Universal Robots URScript: DAS428_958_02_MAR_21_DAS_lado_derecho_jig2.script

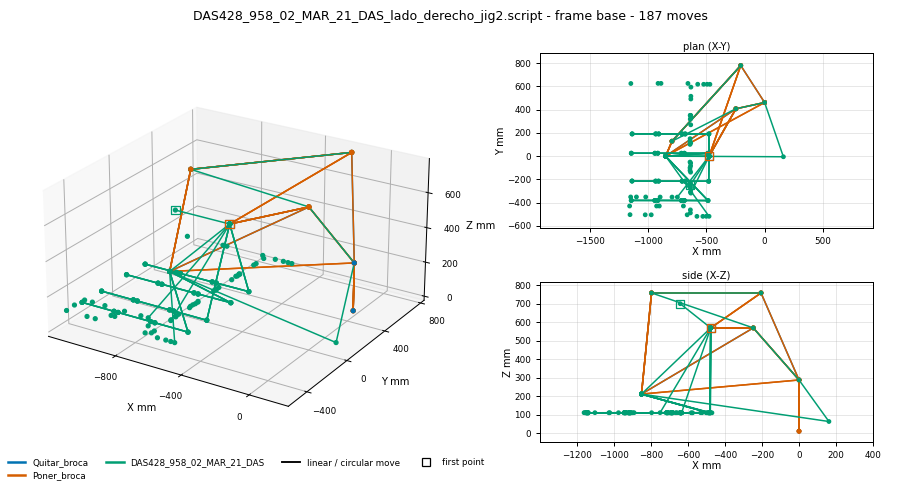
[picture p0: tool path of DAS428_958_02_MAR_21_DAS_lado_derecho_jig2.script in frame base, 187 of 840 moves have a stored position in this frame; points joined in program order, loops and branches not executed]
def DAS428_958_02_MAR_21_DAS_lado_derecho_jig2():
  set_gravity([0.0, 0.0, 9.82])
  set_standard_analog_input_domain(0, 1)
  set_standard_analog_input_domain(1, 1)
  set_tool_analog_input_domain(0, 1)
  set_tool_analog_input_domain(1, 1)
  set_analog_outputdomain(0, 0)
  set_analog_outputdomain(1, 0)
  set_input_actions_to_default()
  set_runstate_standard_digital_outputs([2])
  set_runstate_configurable_digital_outputs([1])
  set_runstate_standard_digital_output_to_value(2, 1)
  set_runstate_configurable_digital_output_to_value(1, 1)
  modbus_add_signal("192.168.10.45", 255, 187, 1, "postrnas_m187", False)
  modbus_set_signal_update_frequency("postrnas_m187", 10)
  modbus_add_signal("192.168.10.45", 255, 289, 1, "ini_cambro_m289", False)
  modbus_set_signal_update_frequency("ini_cambro_m289", 10)
  modbus_add_signal("192.168.10.45", 255, 290, 0, "fin_cambro_m290", False)
  modbus_set_signal_update_frequency("fin_cambro_m290", 10)
  modbus_add_signal("192.168.10.45", 255, 291, 1, "outputbroc_m291", False)
  modbus_set_signal_update_frequency("outputbroc_m291", 10)
  modbus_add_signal("192.168.10.45", 255, 292, 0, "fciclocarr_m292", False)
  modbus_set_signal_update_frequency("fciclocarr_m292", 10)
  modbus_add_signal("192.168.10.45", 255, 7, 1, "avancarrusel_m7", False)
  modbus_set_signal_update_frequency("avancarrusel_m7", 10)
  modbus_add_signal("192.168.10.45", 255, 252, 1, "pose2_m252", False)
  modbus_set_signal_update_frequency("pose2_m252", 10)
  modbus_add_signal("192.168.10.45", 255, 253, 1, "pose3_m253", False)
  modbus_set_signal_update_frequency("pose3_m253", 10)
  modbus_add_signal("192.168.10.45", 255, 254, 1, "pose4_m254", False)
  modbus_set_signal_update_frequency("pose4_m254", 10)
  modbus_add_signal("192.168.10.45", 255, 441, 1, "finciclo_m441", False)
  modbus_set_signal_update_frequency("finciclo_m441", 10)
  modbus_add_signal("192.168.10.45", 255, 442, 1, "finciclo_m442", False)
  modbus_set_signal_update_frequency("finciclo_m442", 10)
  modbus_add_signal("192.168.10.45", 255, 443, 1, "finciclo_m443", False)
  modbus_set_signal_update_frequency("finciclo_m443", 10)
  modbus_add_signal("192.168.10.45", 255, 503, 0, "homecobot_m503", False)
  modbus_set_signal_update_frequency("homecobot_m503", 10)
  modbus_add_signal("192.168.10.45", 255, 288, 1, "cargar_run_m288", False)
  modbus_set_signal_update_frequency("cargar_run_m288", 10)
  modbus_add_signal("192.168.10.45", 255, 287, 0, "desactiver_m288", False)
  modbus_set_signal_update_frequency("desactiver_m288", 10)
  modbus_add_signal("192.168.10.45", 255, 183, 0, "eje7home_m183", False)
  modbus_set_signal_update_frequency("eje7home_m183", 10)
  modbus_add_signal("192.168.10.45", 255, 444, 1, "finciclo_m444", False)
  modbus_set_signal_update_frequency("finciclo_m444", 10)
  modbus_add_signal("192.168.10.45", 255, 381, 0, "pat1_m381", False)
  modbus_set_signal_update_frequency("pat1_m381", 10)
  modbus_add_signal("192.168.10.45", 255, 382, 0, "pat2_m382", False)
  modbus_set_signal_update_frequency("pat2_m382", 10)
  modbus_add_signal("192.168.10.45", 255, 383, 0, "pat3_m383", False)
  modbus_set_signal_update_frequency("pat3_m383", 10)
  modbus_add_signal("192.168.10.45", 255, 384, 0, "pat4_m384", False)
  modbus_set_signal_update_frequency("pat4_m384", 10)
  modbus_add_signal("192.168.10.45", 255, 385, 0, "pat5_m385", False)
  modbus_set_signal_update_frequency("pat5_m385", 10)
  modbus_add_signal("192.168.10.45", 255, 386, 0, "pat6_m386", False)
  modbus_set_signal_update_frequency("pat6_m386", 10)
  modbus_add_signal("192.168.10.45", 255, 387, 0, "pat7_m387", False)
  modbus_set_signal_update_frequency("pat7_m387", 10)
  modbus_add_signal("192.168.10.45", 255, 388, 0, "pat8_m388", False)
  modbus_set_signal_update_frequency("pat8_m388", 10)
  modbus_add_signal("192.168.10.45", 255, 389, 0, "pat9_m389", False)
  modbus_set_signal_update_frequency("pat9_m389", 10)
  modbus_add_signal("192.168.10.45", 255, 390, 0, "pat10_m390", False)
  modbus_set_signal_update_frequency("pat10_m390", 10)
  modbus_add_signal("192.168.10.45", 255, 391, 0, "pat11_m391", False)
  modbus_set_signal_update_frequency("pat11_m391", 10)
  modbus_add_signal("192.168.10.45", 255, 392, 0, "pat12_m392", False)
  modbus_set_signal_update_frequency("pat12_m392", 10)
  modbus_add_signal("192.168.10.45", 255, 401, 0, "inipat1_m401", False)
  modbus_set_signal_update_frequency("inipat1_m401", 10)
  modbus_add_signal("192.168.10.45", 255, 402, 0, "inipat2_m402", False)
  modbus_set_signal_update_frequency("inipat2_m402", 10)
  modbus_add_signal("192.168.10.45", 255, 403, 0, "inipat3_m403", False)
  modbus_set_signal_update_frequency("inipat3_m403", 10)
  modbus_add_signal("192.168.10.45", 255, 404, 0, "inipat4_m404", False)
  modbus_set_signal_update_frequency("inipat4_m404", 10)
  modbus_add_signal("192.168.10.45", 255, 405, 0, "inipat5_m405", False)
  modbus_set_signal_update_frequency("inipat5_m405", 10)
  modbus_add_signal("192.168.10.45", 255, 406, 0, "inipat6_m406", False)
  modbus_set_signal_update_frequency("inipat6_m406", 10)
  modbus_add_signal("192.168.10.45", 255, 407, 0, "inipat7_m407", False)
  modbus_set_signal_update_frequency("inipat7_m407", 10)
  modbus_add_signal("192.168.10.45", 255, 408, 0, "inipat8_m408", False)
  modbus_set_signal_update_frequency("inipat8_m408", 10)
  modbus_add_signal("192.168.10.45", 255, 409, 0, "inipat9_m409", False)
  modbus_set_signal_update_frequency("inipat9_m409", 10)
  modbus_add_signal("192.168.10.45", 255, 410, 0, "inipat10_m410", False)
  modbus_set_signal_update_frequency("inipat10_m410", 10)
  modbus_add_signal("192.168.10.45", 255, 411, 0, "inipat11_m411", False)
  modbus_set_signal_update_frequency("inipat11_m411", 10)
  modbus_add_signal("192.168.10.45", 255, 412, 0, "inipat12_m412", False)
  modbus_set_signal_update_frequency("inipat12_m412", 10)
  modbus_add_signal("192.168.10.45", 255, 430, 0, "modeloDer_m430", False)
  modbus_set_signal_update_frequency("modeloDer_m430", 10)
  modbus_add_signal("192.168.10.45", 255, 380, 1, "mensaje_m380", False)
  modbus_set_signal_update_frequency("mensaje_m380", 10)
  modbus_add_signal("192.168.10.45", 255, 379, 0, "respues_m379", False)
  modbus_set_signal_update_frequency("respues_m379", 10)
  modbus_add_signal("192.168.10.45", 255, 251, 1, "pose1_m251", False)
  modbus_set_signal_update_frequency("pose1_m251", 10)
  modbus_set_runstate_dependent_choice("postrnas_m187",0)
  modbus_set_runstate_dependent_choice("ini_cambro_m289",0)
  modbus_set_runstate_dependent_choice("outputbroc_m291",0)
  modbus_set_runstate_dependent_choice("avancarrusel_m7",0)
  modbus_set_runstate_dependent_choice("pose2_m252",0)
  modbus_set_runstate_dependent_choice("pose3_m253",0)
  modbus_set_runstate_dependent_choice("pose4_m254",0)
  modbus_set_runstate_dependent_choice("finciclo_m441",0)
  modbus_set_runstate_dependent_choice("finciclo_m442",0)
  modbus_set_runstate_dependent_choice("finciclo_m443",0)
  modbus_set_runstate_dependent_choice("cargar_run_m288",0)
  modbus_set_runstate_dependent_choice("finciclo_m444",0)
  modbus_set_runstate_dependent_choice("mensaje_m380",0)
  modbus_set_runstate_dependent_choice("pose1_m251",0)
  set_safety_mode_transition_hardness(1)
  set_tool_communication(False, 115200, 0, 1, 1.5, 3.5)
  set_tool_output_mode(0)
  set_tool_digital_output_mode(0, 1)
  set_tool_digital_output_mode(1, 1)
  set_tool_voltage(0)
  set_tcp(p[4.109330471764039E-4,-0.21829828276152607,0.037994196120996,1.5580092985761962,-0.12546870791316503,0.12120248426608284])
  set_payload(1.5)
  step_count_e0f46a76_adf3_4eac_87f0_1f0dabebea5e = 0
  thread Step_Counter_Thread_08bb6925_5529_4cdb_99f9_8a05e79ee4da():
    while (True):
      step_count_e0f46a76_adf3_4eac_87f0_1f0dabebea5e = step_count_e0f46a76_adf3_4eac_87f0_1f0dabebea5e + 1
      sync()
    end
  end
  run Step_Counter_Thread_08bb6925_5529_4cdb_99f9_8a05e79ee4da()
  global contador=0
  global i_var_1=0
  global Pallet_1_cnt_1=1
  global Pallet_1_cnt=1
  global Line_1=p[0.0,0.0,0.0,0.0,0.0,0.0]
  global Line_2=p[0.0,0.0,0.0,0.0,0.0,0.0]
  global Line_3=p[0.0,0.0,0.0,0.0,0.0,0.0]
  global Line_4=p[-0.2932874787951964,0.3932288129452105,0.013749459185886714,0.019478391032120013,-0.0350876085014595,1.5300278925331599]
  global Line_5=p[0.0,0.0,0.0,0.0,0.0,0.0]
  global Plane_1=p[-0.4357649673792705,0.3571224276764373,-0.011331751409534768,-0.03455953496512708,-0.012487423981114925,3.103751116092306]
  global Plane_2=p[-0.4823864034329737,0.3302516442079689,0.014283714098506706,0.017125077458443067,0.05770060098903715,-2.9134709732588786]
  global Plane_3=p[0.003678615545088639,0.4082921331082374,0.10477407557236007,-2.072177303174012E-4,7.379081343290108E-4,-6.424400645467977E-4]
  global Plane_4=p[-0.4500206307677429,-0.2823718146925442,-0.4767416657426552,0.013278190059218174,0.013334473770785706,1.8479691991032237]
  global Plano_patron1=p[-0.7699005610122596,0.304894434078545,0.0420369514744936,-0.0031270356010209216,1.7180543614697593E-4,-3.508888786211572E-5]
  global Point_13=p[0.0,0.0,0.0,0.0,0.0,0.0]
  global Point_3=p[0.0,0.0,0.0,0.0,0.0,0.0]
  global Point_8=p[0.0,0.0,0.0,0.0,0.0,0.0]
  global Punto_prot_1=p[0.0,0.0,0.0,0.0,0.0,0.0]
  global Punto_seg_der=p[0.23741638234469645,0.3587772222537799,0.42419077585740217,0.818517054876345,1.4216436941132238,1.005041187710707]
  global pisp_958=p[-0.41395442210486977,-0.2082168853247176,0.041553466664982,0.014014788518713659,0.01101911827984854,1.569193423241601]
  rtde_set_watchdog("speed_slider_mask", 10.0, "ignore")
  global Traslacion_p=p[-.641047005341, -.250866212824, .699550653028, 2.557164228531, -1.705634893075, -.146977311260]
  global Traslacion_q=[-0.008123397867477067, -1.6493627997444174, 1.2335318981093104, 0.31142302236535, -5.2726714898139235, -0.002836317283104961]
  global Home2_p=p[-.476229469061, .000000001191, .568736718299, 2.026271312133, -2.392905827360, -.020822003949]
  global Home2_q=[-0.5681294612478887, -2.032770910737735, 1.7176337322759885, 0.3114230223653604, -5.272671489814012, -0.002836317283105849]
  global Home3_p=p[-.850182153427, -.000000001054, .211319941039, -2.029706048810, 2.396843749609, .006593444086]
  global Home3_q=[-0.2508712563283524, -1.32118636682587, 1.7236419957383333, -0.39530717300436535, -4.957384713543316, -0.003346356527782035]
  global Home4_p=p[-.850182153426, -.000000001054, .211319941039, -2.029706048810, 2.396843749609, .006593444086]
  global Home4_q=[-0.25087125632834173, -1.32118636682587, 1.7236419957383335, -0.39530717300436535, -4.957384713543306, -0.003346356527782035]
  global PosicionApagado_p=p[.162342971637, -.004968702407, .063230450635, -1.839175988951, .225343983922, .171657948894]
  global PosicionApagado_q=[1.570738988136085, -1.5704867605983486, 2.609644234392225, 0.2613772922410976, -4.625127484032603, 1.7781079770353217E-5]
  global Precambio_broca_p=p[.000830370305, .461517540512, .287521124194, -.221784750204, -3.131955254916, .000429460883]
  global Precambio_broca_q=[-2.1838225298159477, -2.0964618902985066, 2.243453456263678, -0.13436505871461257, -5.342774534909408, -0.004043449473680738]
  global yendo1_p=p[-.246136658478, .407690142824, .568736718299, -.589365823667, 3.084367220712, .022757599334]
  global yendo1_q=[-1.5957647560042467, -2.0327709107377157, 1.7176337322759783, 0.31142302236534997, -5.272671489813924, -0.002836317283104961]
  global Precam_bro1_p=p[-.795770836809, .128511169110, .757632075886, 1.553391881516, -2.198703969583, -.808866164734]
  global Precam_bro1_q=[-0.42509351308843435, -1.7320527113687803, 1.4689329310980348, -0.39530717300436535, -4.957384713543306, -0.003346356527782035]
  global Precam_bro2_p=p[-.204472177612, .779716277811, .757632075886, -.111446445846, 2.933975892584, 1.018360754732]
  global Precam_bro2_q=[-1.5793151587200072, -1.7320527113687803, 1.4689329310980348, -0.39530717300436535, -4.957384713543306, -0.003346356527782035]
  global Linea1_A_p=p[-.480065223067, -.215566781041, .110154596536, 2.026283817979, -2.392895080548, -.020829635760]
  global Linea1_A_q=[0.12579830563919536, -1.756524695513292, 2.3832893788943412, -0.6314317143827912, -4.58099271090342, -0.0047002730467511356]
  global Linea1_B_p=p[-.683259997836, -.215006380581, .110473377935, 2.026330825697, -2.392937749126, -.020814905630]
  global Linea1_B_q=[0.07860269075896831, -1.433097350639013, 2.069317086211182, -0.6407207629147003, -4.628316962573399, -0.00423059265382264]
  global Linea1_C_p=p[-.708659998696, -.214985847345, .110510820529, 2.026397919151, -2.392909525922, -.020800557194]
  global Linea1_C_q=[0.07508702140477563, -1.3964952588668957, 2.0250632394702635, -0.6330397547175677, -4.631871660537247, -0.004203657105243508]
  global Linea1_D_p=p[-.911541589269, -.214532502479, .110305804030, 2.026334474712, -2.392925442770, -.020895674247]
  global Linea1_D_q=[0.054901387986126586, -1.113040084501037, 1.6299948744075297, -0.5214573164063481, -4.651846197735423, -0.004103335395922336]
  global Linea1_E_p=p[-.936517713267, -.214589312402, .110514758557, 2.026299167222, -2.392914652900, -.020910067647]
  global Linea1_E_q=[0.053256694947611545, -1.0779791152787563, 1.5748557207640133, -0.5014068860788594, -4.65343899925324, -0.0040886755584823575]
  global Linea1_F_p=p[-1.139513888655, -.213880830394, .110127483913, 2.026321929742, -2.392901637414, -.020934114652]
  global Linea1_F_q=[0.04170148606385503, -0.7616832269463547, 1.037979133577118, -0.2808209912067561, -4.664495303417296, -0.0041165609944391335]
  def calculate_point_to_move_towards(feature, direction, position_distance):
    local posDir=[direction[0], direction[1], direction[2]]
    if (norm(posDir) < 1e-6):
      return get_target_waypoint()
    end
    local direction_vector_normalized=normalize(posDir)
    local displacement_pose=p[direction_vector_normalized[0] * position_distance,direction_vector_normalized[1] * position_distance,direction_vector_normalized[2] * position_distance,0,0,0]
    local wanted_displacement_in_base_frame=pose_sub(pose_trans(feature, displacement_pose), feature)
    return pose_add(get_target_waypoint(), wanted_displacement_in_base_frame)
  end
  global Linea2_A_p=p[-.478569784260, .191006236121, .110522539661, 2.026309184484, -2.392844209472, -.020866358396]
  global Linea2_A_q=[-1.0119726055803717, -1.7923449463408154, 2.4087968238915316, -0.622613470734211, -5.718752417482761, 0.0017055247889921077]
  global Linea2_B_p=p[-.681936431684, .191001701528, .110452389888, 2.026254746254, -2.392870981141, -.020856049736]
  global Linea2_B_q=[-0.660932087342812, -1.45042632220569, 2.089702129115615, -0.644100890415773, -5.3678371124098305, -6.551765912714558E-4]
  global Linea2_C_p=p[-.707213860547, .190994877950, .110602621396, 2.026215373389, -2.392855024802, -.020833229234]
  global Linea2_C_q=[-0.6329633221322801, -1.4131450476618888, 2.0452127395946604, -0.63685969915739, -5.339852460491649, -7.508873236439229E-4]
  global Linea2_D_p=p[-.910191818076, .191478760022, .110348317855, 2.026197382673, -2.392838381909, -.020850455695]
  global Linea2_D_q=[-0.47159299446006386, -1.1248659495364315, 1.6481441269090888, -0.5278387233410813, -5.17831767767195, -0.0015522613841945088]
  global Linea2_E_p=p[-.935619999730, .191518537756, .110453838050, 2.026145948950, -2.392831929254, -.020993754227]
  global Linea2_E_q=[-0.45687914266405194, -1.088905585645314, 1.5922022218243828, -0.5079352095297214, -5.1635430614079825, -0.0016331567764398258]
  global Linea2_F_p=p[-1.138394848852, .191499459928, .110212234352, 2.026158962848, -2.392763937758, -.020990642855]
  global Linea2_F_q=[-0.36535169690146674, -0.7732464559921581, 1.0587228640233546, -0.29003791508182974, -5.071546930507635, -0.0021173024104594873]
  global Linea7_A_p=p[-.749560809058, -.351839418109, .110842549516, 3.108416959288, -.375864319326, -.017387250007]
  global Linea7_A_q=[0.03345458497850107, -1.1510417746331125, 1.685959359828983, -0.5377045142036341, -6.168946681556185, -0.005399210077573713]
  global Linea7_B_p=p[-.795370452792, -.351638127396, .110748062148, 3.108426240568, -.375794652077, -.017394126552]
  global Linea7_B_q=[0.031278459806111415, -1.0863508926378662, 1.5866056594622966, -0.5030470097495243, -6.17110138542474, -0.0053959734286266325]
  global Linea8_A_p=p[-.897664645372, -.351420839665, .110405519513, 3.108418537152, -.375848167267, -.017413606898]
  global Linea8_A_q=[0.0274697684633054, -0.9358640938182816, 1.3416002369808222, -0.4084067160106146, -6.174672123664049, -0.005526846744682956]
  global Linea8_B_p=p[-1.021742815617, -.350913421148, .110769725780, 3.108429042178, -.375802310169, -.017313462884]
  global Linea8_B_q=[0.023588010639285104, -0.727028660928073, 0.9730136327156043, -0.24827020482455175, -6.178185664503821, -0.005846159791357053]
  global Linea9_A_p=p[-1.101640143677, -.350630386336, .110828130197, 3.108414048814, -.375882576694, -.017444590769]
  global Linea9_A_q=[0.021544403730552553, -0.5492801598617163, 0.6399908213108159, -0.09279065312938162, -6.179741333586448, -0.006134404310005337]
  global Linea9_B_p=p[-1.151201662491, -.350816300328, .110404811963, 3.108409734650, -.375889963226, -.017367079724]
  global Linea9_B_q=[0.020666902118270467, -0.3678660308533921, 0.2849675943410323, 0.08068312139155243, -6.180088831683512, -0.005949069824949582]
  global Linea10_A_p=p[-.633308011674, -.317691120510, .110994505067, 3.108412257751, -.375924840358, -.017335462218]
  global Linea10_A_q=[-0.015400976327146765, -1.3286836616185038, 1.936773774913373, -0.6125541680104964, -6.2178811871620026, -0.0036320224430834713]
  global Linea10_B_p=p[-.636723959746, -.266696422603, .110313777239, 2.020474030001, -2.393914578871, -.020559556678]
  global Linea10_B_q=[0.1863095606962153, -1.4646980412767157, 2.1071523959293508, -0.6494023099187478, -4.517372761756647, -0.0030763184180990777]
  global Linea11_A_p=p[-.635968117082, -.137768266518, .110291503345, 2.022156502066, -2.396023902726, -.017001304800]
  global Linea11_A_q=[-0.07354604755883543, -1.5471079384277004, 2.1956073198093513, -0.6515202395877564, -4.777150906045714, -0.0016328727799539422]
  global Linea11_B_p=p[-.635823762501, -.083112159886, .110947967545, 2.020383801711, -2.393902625595, -.020556219708]
  global Linea11_B_q=[-0.1908380759122572, -1.5708643495776826, 2.219519946363693, -0.6552069469693311, -4.894453843584338, -5.759924145127826E-4]
  global Linea12_A_p=p[-.635349004319, -.059560123377, .110675436750, 2.020448494290, -2.393915459802, -.020549325419]
  global Linea12_A_q=[-0.2417163087330083, -1.5775265863609773, 2.226737904634896, -0.6557292375944215, -4.945355909075068, -2.7983922817842455E-4]
  global Linea12_B_p=p[-.634712541835, .114180549607, .110553374724, 2.020445364866, -2.393872518012, -.020639369641]
  global Linea12_B_q=[-0.5920002980493377, -1.5626330075993593, 2.212116743928059, -0.656716518252761, -5.2956538993562265, 0.0023497530147947032]
  global Linea13_A_p=p[-.634623456483, .269837596517, .110201600077, 2.020453398687, -2.393912519416, -.020625959570]
  global Linea13_A_q=[-0.8324062816272679, -1.467834151680524, 2.1109901381841176, -0.6517507900808974, -5.53605704845582, 0.004880071949341591]
  global Linea13_B_p=p[-.634042726961, .326314422350, .110496359725, 2.020453146279, -2.393880944182, -.020556436265]
  global Linea13_B_q=[-0.9013131509490719, -1.4220878936638712, 2.0569245075861637, -0.6440785774915501, -5.604971402017175, 0.005892023416525838]
  global Linea14_A_p=p[-.633962563051, .349886895745, .111384319105, 2.020461054934, -2.393837815408, -.020488388436]
  global Linea14_A_q=[-0.9271552684385451, -1.4021744596762797, 2.030901915913411, -0.638246246484969, -5.630828387156736, 0.006335596407090804]
  global Linea14_B_p=p[-.633710645144, .491847819742, .110684020249, 2.020465968208, -2.393853523670, -.020498328553]
  global Linea14_B_q=[-1.0540906694923677, -1.2626852057640106, 1.849914655177884, -0.5986568379003074, -5.757703248039979, 0.008776098960622295]
  global Linea15_A_p=p[-.633318381480, .515440368134, .110157981608, 2.020364155203, -2.393955709596, -.020508500424]
  global Linea15_A_q=[-1.0716567160130523, -1.2377525992845975, 1.8159966720140375, -0.590008690959742, -5.775162769690162, 0.009175048989259693]
  global Linea15_B_p=p[-.632970544234, .593971386241, .110611257026, 2.020441893491, -2.393867996682, -.020560033230]
  global Linea15_B_q=[-1.122474592013197, -1.1525133394351883, 1.6903287270969671, -0.5508046641787523, -5.825981972795807, 0.0105832391144433]
  global Linea16_A_p=p[-.469658501632, .618240146447, .110222995954, -.214451812264, -3.127782132936, -.004019473137]
  global Linea16_A_q=[-1.0558229732465527, -1.3016284898486745, 1.9002200310933528, -0.5927846748758361, -4.220581777772279, 0.011476321502457587]
  global Linea16_B_p=p[-.493719050069, .618586170158, .110182854162, -.214521728939, -3.127775191063, -.003963807283]
  global Linea16_B_q=[-1.0238267857309111, -1.275874279860929, 1.8652664634035965, -0.5834704347683779, -4.1885285819385825, 0.011722546182054927]
  global Linea17_A_p=p[-.523228961738, .618283097935, .110575467666, -.214471054905, -3.127807816993, -.003922935561]
  global Linea17_A_q=[-0.986020922475106, -1.2448369572559947, 1.8212231475782765, -0.570331686133752, -4.150737151059812, 0.011980907174432787]
  global Linea17_B_p=p[-.574504951156, .618780338898, .110128214767, -.214469703842, -3.127802767109, -.003936726452]
  global Linea17_B_q=[-0.9261028235589457, -1.187335623873139, 1.739319222569904, -0.5457499909581429, -4.090780405906422, 0.012429946919677803]
  global Linea18_A_p=p[-.658632612166, .625710002031, .110712740654, -.214452471617, -3.127789736506, -.003965415657]
  global Linea18_A_q=[-0.845178287049178, -1.0844314603972958, 1.5815647493127447, -0.49060909462111013, -4.009765233293088, 0.013074519407750586]
  global Linea18_AB_p=p[-.890202921445, .626113814922, .110875277310, -.214452404345, -3.127789769971, -.003965502225]
  global Linea18_AB_q=[-0.666410313611312, -0.7691628241018513, 1.0473212163579504, -0.27060302401380376, -3.8304915682302414, 0.014782791955626706]
  global Linea18_BA_p=p[-.915681226687, .626148241580, .110663930708, -.214452382992, -3.127789782522, -.003965540155]
  global Linea18_BA_q=[-0.6508504262668842, -0.7263239276067006, 0.9700203563697315, -0.2360215468567155, -3.814840986504011, 0.014958594137021445]
  global Linea18_B_p=p[-1.149588289356, .625184723765, .110393131864, 1.164105535838, -2.905778629907, .010490328627]
  global Linea18_B_q=[-0.6326303647503142, -0.3275146210078148, 0.20111537186222211, 0.13508347000242882, -4.694571332776312, 0.015612052511970474]
  global Linea3_A_p=p[-.486113587685, -.381654790172, .110209853748, -2.029718171558, 2.396836025242, .006539356697]
  global Linea3_A_q=[0.5023501146744431, -1.5361328198955349, 2.1811298091833677, -0.6380602103615596, -4.2045801543318735, 0.0021335806977313965]
  global Linea3_B_p=p[-.689309999510, -.380790560286, .110221298638, -2.029741328186, 2.396866665706, .006544867438]
  global Linea3_B_q=[0.3500483409555937, -1.2996119924085647, 1.897164714326017, -0.5909098707750893, -4.3568479224424745, 0.0011255087267496577]
  global Linea3_C_p=p[-.714729999690, -.381227126176, .110547071161, -2.029776929873, 2.396879295064, .006534577602]
  global Linea3_C_q=[0.33744999495907063, -1.2688250546952826, 1.8544576378801096, -0.5790270771094068, -4.369441028028362, 0.0010604390539933767]
  global Linea3_D_p=p[-.917837219491, -.380541767460, .110221865782, -2.029755394743, 2.396894821329, .006515015900]
  global Linea3_D_q=[0.2571038234470917, -1.0113929982879881, 1.4652198238047056, -0.44729400411425146, -4.449521148440042, 5.150299017975257E-4]
  global Linea3_E_p=p[-.943229998544, -.380750053929, .110259990709, -2.029745434063, 2.396926573302, .006499247846]
  global Linea3_E_q=[0.2498513013118595, -0.9766011167360098, 1.4078530008671004, -0.42473280670143687, -4.4567064172282045, 4.774193732002274E-4]
  global Linea3_F_p=p[-1.146085092422, -.380439604703, .110221400844, -2.029733453251, 2.396965844598, .006565203868]
  global Linea3_F_q=[0.2019713672814234, -0.646294758886178, 0.8226722249789473, -0.16994117112115248, -4.503916586459291, 6.524146887532112E-5]
  global Linea4_A_p=p[-.486108757094, .025046304243, .110758143818, -2.029716299014, 2.396836938000, .006515392677]
  global Linea4_A_q=[-0.6198243103301522, -1.8882999158352325, 2.4675810378541345, -0.5700854657560619, -5.326458533546596, -0.006784361427073726]
  global Linea4_B_p=p[-.689317790597, .025343044299, .110270277143, -2.029778955477, 2.396879909406, .006610652550]
  global Linea4_B_q=[-0.3753982057274481, -1.4863250332384972, 2.127234561670928, -0.6334691626908935, -5.0823254476145046, -0.003953878004303135]
  global Linea4_C_p=p[-.714720878933, .025085639180, .110564947322, -2.029759600612, 2.396870390258, .006543964992]
  global Linea4_C_q=[-0.3574732421871216, -1.4458978723273388, 2.0805072777503337, -0.62720153470989, -5.064395308840017, -0.0037851685217935582]
  global Linea4_D_p=p[-.918062834429, .025352519761, .110171259010, -2.029799128046, 2.396930392653, .006486194650]
  global Linea4_D_q=[-0.2611086455128149, -1.1428166917109337, 1.6724418329476345, -0.5225904730037927, -4.9678804000226116, -0.0028991485058149635]
  global Linea4_E_p=p[-.942590633843, .025362358338, .110649521713, -2.029804551742, 2.396899081770, .006457624074]
  global Linea4_E_q=[-0.25289441014648517, -1.1074268163516194, 1.6172408610903544, -0.5027734532907475, -4.9596442412571164, -0.002849666115224636]
  global Linea4_F_p=p[-1.145809999790, .025560776894, .110408083890, -2.029813008116, 2.396940383966, .006563150563]
  global Linea4_F_q=[-0.20084306122313045, -0.7863624812136436, 1.078794535602439, -0.2855892759874594, -4.907083004154831, -0.00254582608889109]
  global Linea19_A_p=p[-.476993752079, -.517247348420, .110482180983, 3.111546112853, -.391923915264, .008397312856]
  global Linea19_A_q=[0.3663200128941275, -1.4014222930595945, 2.0287178354256366, -0.6180541023023682, -5.826341631139508, -1.5291289902208405E-4]
  global Linea19_B_p=p[-.500828906079, -.517140718168, .110478451867, 3.111546096446, -.391923927944, .008397321867]
  global Linea19_B_q=[0.35160318977889826, -1.372483224500158, 1.9927968502195714, -0.6107942241264501, -5.841051456629851, -4.441148050489119E-4]
  global Linea20_A_p=p[-.530365704390, -.517559293263, .110808466240, 3.111546095803, -.391923919730, .008397321765]
  global Linea20_A_q=[0.33563033058992797, -1.3363269605580115, 1.94574379450221, -0.5995698399171738, -5.857010959106091, -7.866311909552337E-4]
  global Linea20_B_p=p[-.581158312152, -.517498500963, .110403002315, 3.111546108155, -.391923880414, .008397313958]
  global Linea20_B_q=[0.3100718063294732, -1.2734435128638637, 1.862269700997377, -0.5783990031154378, -5.8825402788566326, -0.0013910864741042417]
  global Linea21_A_p=p[-.665124494580, -.504210865882, .110600214775, 3.111546096026, -.391923862954, .008397317428]
  global Linea21_A_q=[0.2573690543360489, -1.1776890584644226, 1.7249145049026704, -0.5352634869878585, -5.935170767510868, -0.002981287852510839]
  global Linea21_AB_p=p[-.974251236041, -.504210865628, .110800066306, 3.111546114034, -.391923818122, .008397307719]
  global Linea21_AB_q=[0.1799298970176908, -0.7275076895770098, 0.9726424894081029, -0.22955136462346193, -6.011907604967895, -0.006694782410928468]
  global Linea21_BA_p=p[-1.025948854959, -.504193334254, .110365518030, 3.111461951708, -.391950297460, .007971986720]
  global Linea21_BA_q=[0.1711561465100031, -0.6245380104555593, 0.7826065934061077, -0.14219863176293934, -6.020415742618897, -0.00727529467707555]
  global Linea21_B_p=p[-1.156707649875, -.503072794545, .110552345697, -2.509967435901, 1.875250959640, .002018781675]
  global Linea21_B_q=[0.24820218748779244, -0.5254029363972528, 0.5900463054518754, -0.04848122613311023, -4.910307707512297, -0.005929498886956708]
  global Linea22_A_p=p[-.637632433174, -.487982976479, .110979882815, 3.111546090028, -.391923816497, .008397315714]
  global Linea22_A_q=[0.24472934312467132, -1.2243225409022536, 1.7920552918632602, -0.5553129495014248, -5.947844161109764, -0.0034535219061346822]
  global Linea22_B_p=p[-.637632431354, -.461705375702, .110442752941, 3.111546036492, -.391923771717, .008397328631]
  global Linea22_B_q=[0.20717345223233252, -1.241126788140571, 1.8170870077379373, -0.5619896731518628, -5.985409130317459, -0.0050445535333150104]
  global Linea23_A_p=p[-.637534615339, -.308489261992, .110677052130, 3.111545937941, -.391923740021, .008397338509]
  global Linea23_A_q=[-0.028811057420131903, -1.3103407381530268, 1.9122910134814681, -0.5347248377646263, -6.221285712923422, -0.05854924353866764]
  global Linea23_B_p=p[-.640733962739, -.257360958137, .110320484628, -1.919417494801, 2.483289836721, .006037999405]
  global Linea23_B_q=[0.1905486224517663, -1.450436264205365, 2.0857635636442016, -0.6270384051172089, -4.427102446372631, -1.2154783732398755E-4]
  global Linea24_A_p=p[-.640733961490, -.233284408478, .110638871698, -1.919417552760, 2.483289783731, .006038056909]
  global Linea24_A_q=[0.14545722065475164, -1.4688531178545041, 2.1062141334115556, -0.629125928981761, -4.472191088464225, -5.194241954580292E-4]
  global Linea24_B_p=p[-.640733960275, -.122850233085, .110748525345, -1.919417597211, 2.483289752526, .006038102658]
  global Linea24_B_q=[-0.07605491895077954, -1.5353858090675878, 2.1786254928410287, -0.6349982171419359, -4.693686238133267, -0.0024004120313705357]
  global Linea25_A_p=p[-.640733959025, -.099756217052, .110149053398, -1.919417622933, 2.483289733447, .006038127253]
  global Linea25_A_q=[-0.1244406410731358, -1.544441361062633, 2.189369992241023, -0.6366292245286829, -4.742070057375175, -0.0028048012168682135]
  global Linea25_B_p=p[-.640733958354, -.050488778220, .110217684856, -1.919417690989, 2.483289674763, .006038178959]
  global Linea25_B_q=[-0.2283127239691316, -1.5597473241762696, 2.204914426396905, -0.6366747472205034, -4.845933707721189, -0.003691692902822119]
  global Linea26_A_p=p[-.640547506113, .101329564039, .110865193067, -1.919417715349, 2.483289689335, .006038198474]
  global Linea26_A_q=[-0.5332933914937019, -1.5549547991705772, 2.1986195220763918, -0.6339933161425408, -5.150899742746004, -0.006567092346116965]
  global Linea26_B_p=p[-.640680925269, .126812188772, .110399195482, -1.919417776128, 2.483289636172, .006038228077]
  global Linea26_B_q=[-0.5793189919827881, -1.5454213815793807, 2.1898401188412677, -0.6344739078467976, -5.196927100374702, -0.007060981198389271]
  global Linea27_A_p=p[-.640020451439, .150733100880, .110213160527, -1.919417813264, 2.483289585399, .006038241789]
  global Linea27_A_q=[-0.6217233925628083, -1.536230558235598, 2.180685216451952, -0.6342282470711922, -5.2393319968885415, -0.007541218547958195]
  global Linea27_B_p=p[-.638705853179, .318073094658, .110644167614, .116299088145, 3.121658150077, .005213984395]
  global Linea27_B_q=[-0.5302181957807237, -1.311893423219579, 1.9124676839697672, -0.5889762150838447, -3.75724236079801, -0.005733470438864963]
  global Linea28_B_p=p[-.638705854413, .351254438579, .110847636331, .116299139192, 3.121658163812, .005213903305]
  global Linea28_B_q=[-0.5749160295300664, -1.298447915414732, 1.8940103653434506, -0.5845949761528715, -3.801930405986168, -0.006576175916428895]
  global Linea29_A_p=p[-.697641532877, -.428593360272, .109990008742, -2.801724319039, 1.417160453684, .007198341972]
  global Linea29_A_q=[0.23527656453246326, -1.2789397769027335, 1.8687632760476625, -0.5784646150523693, -5.271258681648637, -0.008392583459158942]
  global Linea29_AB_p=p[-.904922459205, -.428636744368, .110456720257, -2.801724313385, 1.417160441963, .007198353879]
  global Linea29_AB_q=[0.17841388372429012, -1.0033716864184807, 1.4509125680551742, -0.43568055422700613, -5.327850178749621, -0.009190677590165564]
  global Linea29_BA_p=p[-.927926651083, -.428699716140, .110396892952, -2.803374774073, 1.417906295507, .010979680109]
  global Linea29_BA_q=[0.1737614027292249, -0.9719074952973319, 1.3997777298545344, -0.41899622204942855, -5.332520268083923, -0.0092330916124439]
  global Linea29_B_p=p[-1.160230525221, -.428650841833, .110797243179, -2.801724280945, 1.417160425039, .007198392254]
  global Linea29_B_q=[0.1368429869194676, -0.5546997699196048, 0.6476482713797873, -0.08061893151237864, -5.368496825996519, -0.009905759515234536]
  global Dejar_broca_p=p[.000823895285, .461515686418, .010824983886, -.221812507768, -3.131977618886, .000372128741]
  global Dejar_broca_q=[-2.183487269545523, -1.7626289818446779, 2.619089631151862, -0.8448915610823917, -5.34389996121201, -0.0023222697552238714]
  def Quitar_broca():
    $ 5362 "Quitar_broca" "noBreak"
    $ 5363 "Quitar_broca"
    $ 5364 "barrenos_hechos≔barrenos_hechos+1"
    global barrenos_hechos=barrenos_hechos+1
    $ 5371 "If barrenos_hechos≟14 or cambiar_broca≟ True "
    if (barrenos_hechos == 14  or  cambiar_broca ==   True  ):
      $ 5372 "'Codigo de quitar broca'"
      # 'Codigo de quitar broca'
      $ 5373 "MoveL"
      $ 5374 "Direction: Base Z+"
      global move_thread_flag_5374=0
      thread move_thread_5374():
        enter_critical
        move_thread_flag_5374 = 1
        local towardsPos=calculate_point_to_move_towards(p[0.0,0.0,0.0,0.0,0.0,0.0], [0.0,0.0,1.0], 0.05)
        movel(towardsPos, a=1.2, v=0.25)
        move_thread_flag_5374 = 2
        exit_critical
      end
      move_thread_flag_5374 = 0
      move_thread_han_5374 = run move_thread_5374()
      while (True):
        sleep(1.0E-10)
        if (move_thread_flag_5374 > 1):
          join move_thread_han_5374
          $ 5375 "Until (distance)"
          break
        end
        sync()
      end
      $ 5376 "If eje7≟2"
      if (eje7 == 2):
        $ 5377 "Home2" "breakAfter"
        movel(Home2_p, a=1.2, v=0.25)
        $ 5378 "yendo1" "breakAfter"
        movel(yendo1_p, a=1.2, v=0.25)
      end
      $ 5379 "If eje7≟3"
      if (eje7 == 3):
        $ 5380 "Home3" "breakAfter"
        movel(Home3_p, a=1.2, v=0.25)
        $ 5381 "Precam_bro1" "breakAfter"
        movel(Precam_bro1_p, a=1.2, v=0.25)
        $ 5382 "Precam_bro2" "breakAfter"
        movel(Precam_bro2_p, a=1.2, v=0.25)
      end
      $ 5383 "Precambio_broca" "breakAfter"
      movel(Precambio_broca_p, a=1.2, v=0.25)
      $ 5384 "Dejar_broca" "breakAfter"
      movel(Dejar_broca_p, a=0.1, v=0.09)
      $ 5385 "Set outputbroc_m291=Encender"
      modbus_set_output_signal("outputbroc_m291", True)
      $ 5386 "Wait: 2.0"
      sleep(2.0)
      $ 5388 "Wait: 2.0"
      sleep(2.0)
      $ 5389 "Set outputbroc_m291=Apagar"
      modbus_set_output_signal("outputbroc_m291", False)
      $ 5390 "Wait: 0.5"
      sleep(0.5)
      $ 5391 "Wait fciclocarr_m292=LO"
      while (modbus_get_signal_status("fciclocarr_m292") == True):
        sync()
      end
      $ 5392 "Wait: 0.5"
      sleep(0.5)
      $ 5394 "MoveL"
      $ 5395 "Precambio_broca" "breakAfter"
      movel(Precambio_broca_p, a=0.1, v=0.09)
      $ 5396 "Set avancarrusel_m7=Encender"
      modbus_set_output_signal("avancarrusel_m7", True)
      $ 5397 "Wait: 2.0"
      sleep(2.0)
      $ 5398 "Set avancarrusel_m7=Apagar"
      modbus_set_output_signal("avancarrusel_m7", False)
      $ 5399 "Wait: 0.1"
      sleep(0.1)
    end
  end
  def Poner_broca():
    $ 5400 "Poner_broca" "noBreak"
    $ 5401 "Poner_broca"
    $ 5402 "If cambiar_broca≟ True  or iniciando_prog≟ True "
    if (cambiar_broca ==   True    or  iniciando_prog ==   True  ):
      $ 5403 "'Codigo de poner broca'"
      # 'Codigo de poner broca'
      $ 5404 "Set ini_cambro_m289=Apagar"
      modbus_set_output_signal("ini_cambro_m289", False)
      $ 5405 "MoveL"
      $ 5406 "If eje7≟2 and iniciando_prog≟ True "
      if (eje7 == 2  and  iniciando_prog ==   True  ):
        $ 5407 "Home2" "breakAfter"
        movel(Home2_p, a=1.2, v=0.25)
        $ 5408 "yendo1" "breakAfter"
        movel(yendo1_p, a=1.2, v=0.25)
      end
      $ 5409 "If eje7≟3 and iniciando_prog≟ True "
      if (eje7 == 3  and  iniciando_prog ==   True  ):
        $ 5410 "Home3" "breakAfter"
        movel(Home3_p, a=1.2, v=0.25)
        $ 5411 "Precam_bro1" "breakAfter"
        movel(Precam_bro1_p, a=1.2, v=0.25)
        $ 5412 "Precam_bro2" "breakAfter"
        movel(Precam_bro2_p, a=1.2, v=0.25)
      end
      $ 5413 "Precambio_broca" "breakAfter"
      movel(Precambio_broca_p, a=1.2, v=0.25)
      $ 5414 "Popup: Cambia a las siguientes brocas"
      popup("Cambia a las siguientes brocas", "Advertencia", True, False, blocking=True)
      $ 5415 "Dejar_broca" "breakAfter"
      movel(Dejar_broca_p, a=0.1, v=0.09)
      $ 5416 "Set ini_cambro_m289=Encender"
      modbus_set_output_signal("ini_cambro_m289", True)
      $ 5417 "Wait: 2.0"
      sleep(2.0)
      $ 5419 "Wait: 2.0"
      sleep(2.0)
      $ 5420 "Set ini_cambro_m289=Apagar"
      modbus_set_output_signal("ini_cambro_m289", False)
      $ 5421 "Wait: 0.5"
      sleep(0.5)
      $ 5422 "Wait fciclocarr_m292=LO"
      while (modbus_get_signal_status("fciclocarr_m292") == True):
        sync()
      end
      $ 5423 "Wait: 0.5"
      sleep(0.5)
      $ 5425 "MoveL"
      $ 5426 "Precambio_broca" "breakAfter"
      movel(Precambio_broca_p, a=0.1, v=0.09)
      $ 5427 "If eje7≟2"
      if (eje7 == 2):
        $ 5428 "yendo1" "breakAfter"
        movel(yendo1_p, a=1.2, v=0.25)
        $ 5429 "Home2" "breakAfter"
        movel(Home2_p, a=1.2, v=0.25)
      end
      $ 5430 "If eje7≟3"
      if (eje7 == 3):
        $ 5431 "Precam_bro2" "breakAfter"
        movel(Precam_bro2_p, a=1.2, v=0.25)
        $ 5432 "Precam_bro1" "breakAfter"
        movel(Precam_bro1_p, a=1.2, v=0.25)
        $ 5433 "Home3" "breakAfter"
        movel(Home3_p, a=1.2, v=0.25)
      end
      $ 5434 "barrenos_hechos≔0"
      global barrenos_hechos=0
      $ 5435 "iniciando_prog≔ False "
      global iniciando_prog=  False
      $ 5436 "cambiar_broca≔ False "
      global cambiar_broca=  False
    end
    $ 5437 "If barrenos_hechos≟14"
    if (barrenos_hechos == 14):
      $ 5438 "If cambiar_broca≟ False "
      if (cambiar_broca ==   False  ):
        $ 5439 "'Codigo de poner broca'"
        # 'Codigo de poner broca'
        $ 5440 "Set ini_cambro_m289=Apagar"
        modbus_set_output_signal("ini_cambro_m289", False)
        $ 5441 "MoveL"
        $ 5442 "Precambio_broca" "breakAfter"
        movel(Precambio_broca_p, a=1.2, v=0.25)
        $ 5443 "Dejar_broca" "breakAfter"
        movel(Dejar_broca_p, a=0.1, v=0.09)
        $ 5444 "Set ini_cambro_m289=Encender"
        modbus_set_output_signal("ini_cambro_m289", True)
        $ 5445 "Wait: 2.0"
        sleep(2.0)
        $ 5447 "Wait: 2.0"
        sleep(2.0)
        $ 5448 "Set ini_cambro_m289=Apagar"
        modbus_set_output_signal("ini_cambro_m289", False)
        $ 5449 "Wait: 0.5"
        sleep(0.5)
        $ 5450 "Wait fciclocarr_m292=LO"
        while (modbus_get_signal_status("fciclocarr_m292") == True):
          sync()
        end
        $ 5451 "Wait: 0.5"
        sleep(0.5)
        $ 5453 "MoveL"
        $ 5454 "Precambio_broca" "breakAfter"
        movel(Precambio_broca_p, a=0.1, v=0.09)
        $ 5455 "If eje7≟2"
        if (eje7 == 2):
          $ 5456 "yendo1" "breakAfter"
          movel(yendo1_p, a=1.2, v=0.25)
          $ 5457 "Home2" "breakAfter"
          movel(Home2_p, a=1.2, v=0.25)
        end
        $ 5458 "If eje7≟3"
        if (eje7 == 3):
          $ 5459 "Precam_bro2" "breakAfter"
          movel(Precam_bro2_p, a=1.2, v=0.25)
          $ 5460 "Precam_bro1" "breakAfter"
          movel(Precam_bro1_p, a=1.2, v=0.25)
          $ 5461 "Home3" "breakAfter"
          movel(Home3_p, a=1.2, v=0.25)
        end
        $ 5462 "barrenos_hechos≔0"
        global barrenos_hechos=0
        $ 5463 "iniciando_prog≔ False "
        global iniciando_prog=  False
        $ 5464 "cambiar_broca≔ False "
        global cambiar_broca=  False
      else:
        $ 5465 "Else" "noBreak"
        $ 5466 "'Codigo de poner broca'"
        # 'Codigo de poner broca'
        $ 5467 "Set ini_cambro_m289=Apagar"
        modbus_set_output_signal("ini_cambro_m289", False)
        $ 5468 "MoveL"
        $ 5469 "Precambio_broca" "breakAfter"
        movel(Precambio_broca_p, a=1.2, v=0.25)
        $ 5470 "Popup: Cambia a las siguientes brocas"
        popup("Cambia a las siguientes brocas", "Advertencia", True, False, blocking=True)
        $ 5471 "Dejar_broca" "breakAfter"
        movel(Dejar_broca_p, a=0.1, v=0.09)
        $ 5472 "Set ini_cambro_m289=Encender"
        modbus_set_output_signal("ini_cambro_m289", True)
        $ 5473 "Wait: 2.0"
        sleep(2.0)
        $ 5475 "Wait: 2.0"
        sleep(2.0)
        $ 5476 "Set ini_cambro_m289=Apagar"
        modbus_set_output_signal("ini_cambro_m289", False)
        $ 5477 "Wait: 0.5"
        sleep(0.5)
        $ 5478 "Wait fciclocarr_m292=LO"
        while (modbus_get_signal_status("fciclocarr_m292") == True):
          sync()
        end
        $ 5479 "Wait: 0.5"
        sleep(0.5)
        $ 5481 "MoveL"
        $ 5482 "Precambio_broca" "breakAfter"
        movel(Precambio_broca_p, a=0.1, v=0.09)
        $ 5483 "If eje7≟2"
        if (eje7 == 2):
          $ 5484 "yendo1" "breakAfter"
          movel(yendo1_p, a=1.2, v=0.25)
          $ 5485 "Home2" "breakAfter"
          movel(Home2_p, a=1.2, v=0.25)
        end
        $ 5486 "If eje7≟3"
        if (eje7 == 3):
          $ 5487 "Precam_bro2" "breakAfter"
          movel(Precam_bro2_p, a=1.2, v=0.25)
          $ 5488 "Precam_bro1" "breakAfter"
          movel(Precam_bro1_p, a=1.2, v=0.25)
          $ 5489 "Home3" "breakAfter"
          movel(Home3_p, a=1.2, v=0.25)
        end
        $ 5490 "barrenos_hechos≔0"
        global barrenos_hechos=0
        $ 5491 "iniciando_prog≔ False "
        global iniciando_prog=  False
        $ 5492 "cambiar_broca≔ False "
        global cambiar_broca=  False
      end
    end
  end
  while (True):
    $ 1 "Robot Program"
    $ 2 "Variables"
    $ 3 "bajada_broca≔p[0,0,-0.008,0,0,0]"
    global bajada_broca=p[0,0,-0.008,0,0,0]
    $ 4 "barrenos_menos1≔0"
    global barrenos_menos1=0
    $ 5 "barreno_actual≔0"
    global barreno_actual=0
    $ 6 "posicion≔p[0,0,300,0,0,0]"
    global posicion=p[0,0,300,0,0,0]
    $ 7 "cambiar_broca≔ False "
    global cambiar_broca=  False
    $ 8 "barrenos_hechos≔0"
    global barrenos_hechos=0
    $ 9 "eje7≔0"
    global eje7=0
    $ 10 "Wait: 0.5"
    sleep(0.5)
    $ 11 "Home"
    $ 12 "Wait: 0.3"
    sleep(0.3)
    $ 13 "MoveL"
    $ 14 "Traslacion" "breakAfter"
    movel(Traslacion_p, a=1.2, v=0.25)
    $ 15 "Home2" "breakAfter"
    movel(Home2_p, a=1.2, v=0.25)
    $ 16 "Home3" "breakAfter"
    movel(Home3_p, a=1.2, v=0.25)
    $ 17 "Home4" "breakAfter"
    movel(Home4_p, a=1.2, v=0.25)
    $ 18 "PosicionApagado" "breakAfter"
    movel(PosicionApagado_p, a=1.2, v=0.25)
    $ 19 "Precambio_broca" "breakAfter"
    movel(Precambio_broca_p, a=1.2, v=0.25)
    $ 20 "yendo1" "breakAfter"
    movel(yendo1_p, a=1.2, v=0.25)
    $ 21 "Precam_bro1" "breakAfter"
    movel(Precam_bro1_p, a=1.2, v=0.25)
    $ 22 "Precam_bro2" "breakAfter"
    movel(Precam_bro2_p, a=1.2, v=0.25)
    $ 23 "Home"
    movej([1.5707389881360854, -1.5704867605983486, 2.609644234392224, 0.2613772922410976, -4.625127484032603, 1.7781079770351482E-5], a=1.3962634015954636, v=1.0471975511965976)
    $ 31 "Wait: 0.3"
    sleep(0.3)
    $ 32 "iniciando_prog≔ True "
    global iniciando_prog=  True
    $ 33 "Call Poner_broca"
    Poner_broca()
    $ 34 "Posicion2"
    $ 35 "Inicio"
    $ 36 "eje7≔2"
    global eje7=2
    $ 37 "MoveL"
    $ 38 "Home2" "breakAfter"
    movel(Home2_p, a=1.2, v=0.25)
    $ 39 "SeatTracks"
    $ 40 "Broca_1"
    $ 41 "Linea1"
    $ 42 "Marcar_puntos"
    $ 43 "MoveL"
    $ 44 "Home2" "breakAfter"
    movel(Home2_p, a=0.5, v=0.1)
    $ 52 "Linea1_A" "breakAfter"
    movel(Linea1_A_p, a=0.5, v=0.1)
    $ 53 "Linea1_B" "breakAfter"
    movel(Linea1_B_p, a=0.5, v=0.1)
    $ 54 "Linea1_C" "breakAfter"
    movel(Linea1_C_p, a=0.5, v=0.1)
    $ 55 "Linea1_D" "breakAfter"
    movel(Linea1_D_p, a=0.5, v=0.1)
    $ 56 "Linea1_E" "breakAfter"
    movel(Linea1_E_p, a=0.5, v=0.1)
    $ 57 "Linea1_F" "breakAfter"
    movel(Linea1_F_p, a=0.5, v=0.1)
    $ 58 "AB"
    $ 59 "'desbaste_inicial'"
    # 'desbaste_inicial'
    $ 60 "bajada_broca≔p[0,0,-0.008,0,0,0]"
    global bajada_broca=p[0,0,-0.008,0,0,0]
    $ 61 "barrenos_menos1≔8"
    global barrenos_menos1=8
    $ 62 "barreno_actual≔0"
    global barreno_actual=0
    $ 63 "Loop barreno_actual≤barrenos_menos1"
    while (barreno_actual <= barrenos_menos1):
      $ 64 "Perforacion"
      $ 65 "MoveL"
      $ 66 "internos≔interpolate_pose(Linea1_A, Linea1_B, barreno_actual/barrenos_menos1)"
      global internos= interpolate_pose (Linea1_A_p, Linea1_B_p, barreno_actual/barrenos_menos1)
      $ 67 "internos" "breakAfter"
      movel(internos, a=0.5, v=0.1)
      $ 68 "'desbaste_inicial'"
      # 'desbaste_inicial'
      $ 69 "bajada_broca≔p[0,0,-0.008,0,0,0]"
      global bajada_broca=p[0,0,-0.008,0,0,0]
      $ 70 "bajada≔p[0,0,0.008,0,0,0]"
      global bajada=p[0,0,0.008,0,0,0]
      $ 71 "Direction: Base Z-"
      global move_thread_flag_71=0
      thread move_thread_71():
        enter_critical
        move_thread_flag_71 = 1
        local towardsPos=calculate_point_to_move_towards(p[0.0,0.0,0.0,0.0,0.0,0.0], [0.0,0.0,-1.0], 0.076)
        movel(towardsPos, a=0.035, v=0.03)
        move_thread_flag_71 = 2
        exit_critical
      end
      move_thread_flag_71 = 0
      move_thread_han_71 = run move_thread_71()
      while (True):
        sleep(1.0E-10)
        if (move_thread_flag_71 > 1):
          join move_thread_han_71
          $ 72 "Until (distance)"
          break
        end
        sync()
      end
      $ 73 "Popup: punto contacto alanzdo"
      popup("punto contacto alanzdo", "Mensaje", False, False, blocking=True)
      $ 74 "Direction: Base Z+"
      global move_thread_flag_74=0
      thread move_thread_74():
        enter_critical
        move_thread_flag_74 = 1
        local towardsPos=calculate_point_to_move_towards(p[0.0,0.0,0.0,0.0,0.0,0.0], [0.0,0.0,1.0], 0.002)
        movel(towardsPos, a=0.005, v=0.003)
        move_thread_flag_74 = 2
        exit_critical
      end
      move_thread_flag_74 = 0
      move_thread_han_74 = run move_thread_74()
      while (True):
        sleep(1.0E-10)
        if (move_thread_flag_74 > 1):
          join move_thread_han_74
          $ 75 "Until (distance)"
          break
        end
        sync()
      end
      $ 76 "Wait: 0.3"
      sleep(0.3)
      $ 77 "Set CO[1]=Encender"
      set_configurable_digital_out(1, True)
      $ 78 "Wait: 0.3"
      sleep(0.3)
      $ 79 "Loop 3 times"
      Loop_39 = 0
      while (Loop_39 < 3):
        $ 80 "bajar≔pose_add(get_actual_tcp_pose(), bajada_broca)"
        global bajar= pose_add ( get_actual_tcp_pose (), bajada_broca)
        $ 81 "bajar" "breakAfter"
        movel(bajar, a=0.005, v=0.001)
        $ 82 "subir≔pose_sub(get_actual_tcp_pose(), bajada_broca)"
        global subir= pose_sub ( get_actual_tcp_pose (), bajada_broca)
        $ 83 "subir" "breakAfter"
        movel(subir, a=0.01, v=0.005)
        $ 84 "bajada_broca≔pose_sub(bajada_broca, bajada)"
        global bajada_broca= pose_sub (bajada_broca, bajada)
        Loop_39 = Loop_39 + 1
      end
      $ 85 "Direction: Base Z+"
      global move_thread_flag_85=0
      thread move_thread_85():
        enter_critical
        move_thread_flag_85 = 1
        local towardsPos=calculate_point_to_move_towards(p[0.0,0.0,0.0,0.0,0.0,0.0], [0.0,0.0,1.0], 0.06)
        movel(towardsPos, a=0.035, v=0.03)
        move_thread_flag_85 = 2
        exit_critical
      end
      move_thread_flag_85 = 0
      move_thread_han_85 = run move_thread_85()
      while (True):
        sleep(1.0E-10)
        if (move_thread_flag_85 > 1):
          join move_thread_han_85
          $ 86 "Until (distance)"
          break
        end
        sync()
      end
      $ 87 "Set CO[1]=Apagar"
      set_configurable_digital_out(1, False)
      $ 88 "barreno_actual≔barreno_actual+1"
      global barreno_actual=barreno_actual+1
      $ 89 "Call Quitar_broca"
      Quitar_broca()
      $ 90 "Call Poner_broca"
      Poner_broca()
    end
    $ 91 "CD"
    $ 92 "'desbaste_inicial'"
    # 'desbaste_inicial'
    $ 93 "bajada_broca≔p[0,0,-0.008,0,0,0]"
    global bajada_broca=p[0,0,-0.008,0,0,0]
    $ 94 "barrenos_menos1≔8"
    global barrenos_menos1=8
    $ 95 "barreno_actual≔0"
    global barreno_actual=0
    $ 96 "Loop barreno_actual≤barrenos_menos1"
    while (barreno_actual <= barrenos_menos1):
      $ 97 "Perforacion"
      $ 98 "MoveL"
      $ 99 "internos≔interpolate_pose(Linea1_C, Linea1_D, barreno_actual/barrenos_menos1)"
      global internos= interpolate_pose (Linea1_C_p, Linea1_D_p, barreno_actual/barrenos_menos1)
      $ 100 "internos" "breakAfter"
      movel(internos, a=0.5, v=0.1)
      $ 101 "'desbaste_inicial'"
      # 'desbaste_inicial'
      $ 102 "bajada_broca≔p[0,0,-0.008,0,0,0]"
      global bajada_broca=p[0,0,-0.008,0,0,0]
      $ 103 "bajada≔p[0,0,0.008,0,0,0]"
      global bajada=p[0,0,0.008,0,0,0]
      $ 104 "Direction: Base Z-"
      global move_thread_flag_104=0
      thread move_thread_104():
        enter_critical
        move_thread_flag_104 = 1
        local towardsPos=calculate_point_to_move_towards(p[0.0,0.0,0.0,0.0,0.0,0.0], [0.0,0.0,-1.0], 0.076)
        movel(towardsPos, a=0.035, v=0.03)
        move_thread_flag_104 = 2
        exit_critical
      end
      move_thread_flag_104 = 0
      move_thread_han_104 = run move_thread_104()
      while (True):
        sleep(1.0E-10)
        if (move_thread_flag_104 > 1):
          join move_thread_han_104
          $ 105 "Until (distance)"
          break
        end
        sync()
      end
      $ 106 "Popup: punto contacto alanzdo"
      popup("punto contacto alanzdo", "Mensaje", False, False, blocking=True)
      $ 107 "Direction: Base Z+"
      global move_thread_flag_107=0
      thread move_thread_107():
        enter_critical
        move_thread_flag_107 = 1
        local towardsPos=calculate_point_to_move_towards(p[0.0,0.0,0.0,0.0,0.0,0.0], [0.0,0.0,1.0], 0.002)
        movel(towardsPos, a=0.005, v=0.003)
        move_thread_flag_107 = 2
        exit_critical
      end
      move_thread_flag_107 = 0
      move_thread_han_107 = run move_thread_107()
      while (True):
        sleep(1.0E-10)
        if (move_thread_flag_107 > 1):
          join move_thread_han_107
          $ 108 "Until (distance)"
          break
        end
        sync()
      end
      $ 109 "Wait: 0.3"
      sleep(0.3)
      $ 110 "Set CO[1]=Encender"
      set_configurable_digital_out(1, True)
      $ 111 "Wait: 0.3"
      sleep(0.3)
      $ 112 "Loop 3 times"
      Loop_56 = 0
      while (Loop_56 < 3):
        $ 113 "bajar≔pose_add(get_actual_tcp_pose(), bajada_broca)"
        global bajar= pose_add ( get_actual_tcp_pose (), bajada_broca)
        $ 114 "bajar" "breakAfter"
        movel(bajar, a=0.005, v=0.001)
        $ 115 "subir≔pose_sub(get_actual_tcp_pose(), bajada_broca)"
        global subir= pose_sub ( get_actual_tcp_pose (), bajada_broca)
        $ 116 "subir" "breakAfter"
        movel(subir, a=0.01, v=0.005)
        $ 117 "bajada_broca≔pose_sub(bajada_broca, bajada)"
        global bajada_broca= pose_sub (bajada_broca, bajada)
        Loop_56 = Loop_56 + 1
      end
      $ 118 "Direction: Base Z+"
      global move_thread_flag_118=0
      thread move_thread_118():
        enter_critical
        move_thread_flag_118 = 1
        local towardsPos=calculate_point_to_move_towards(p[0.0,0.0,0.0,0.0,0.0,0.0], [0.0,0.0,1.0], 0.06)
        movel(towardsPos, a=0.035, v=0.03)
        move_thread_flag_118 = 2
        exit_critical
      end
      move_thread_flag_118 = 0
      move_thread_han_118 = run move_thread_118()
      while (True):
        sleep(1.0E-10)
        if (move_thread_flag_118 > 1):
          join move_thread_han_118
          $ 119 "Until (distance)"
          break
        end
        sync()
      end
      $ 120 "Set CO[1]=Apagar"
      set_configurable_digital_out(1, False)
      $ 121 "barreno_actual≔barreno_actual+1"
      global barreno_actual=barreno_actual+1
      $ 122 "Call Quitar_broca"
      Quitar_broca()
      $ 123 "Call Poner_broca"
      Poner_broca()
    end
    $ 124 "EF"
    $ 125 "'desbaste_inicial'"
    # 'desbaste_inicial'
    $ 126 "bajada_broca≔p[0,0,-0.008,0,0,0]"
    global bajada_broca=p[0,0,-0.008,0,0,0]
    $ 127 "barrenos_menos1≔8"
    global barrenos_menos1=8
    $ 128 "barreno_actual≔0"
    global barreno_actual=0
    $ 129 "Loop barreno_actual≤barrenos_menos1"
    while (barreno_actual <= barrenos_menos1):
      $ 130 "Perforacion"
      $ 131 "MoveL"
      $ 132 "internos≔interpolate_pose(Linea1_E, Linea1_F, barreno_actual/barrenos_menos1)"
      global internos= interpolate_pose (Linea1_E_p, Linea1_F_p, barreno_actual/barrenos_menos1)
      $ 133 "internos" "breakAfter"
      movel(internos, a=0.5, v=0.1)
      $ 134 "'desbaste_inicial'"
      # 'desbaste_inicial'
      $ 135 "bajada_broca≔p[0,0,-0.008,0,0,0]"
      global bajada_broca=p[0,0,-0.008,0,0,0]
      $ 136 "bajada≔p[0,0,0.008,0,0,0]"
      global bajada=p[0,0,0.008,0,0,0]
      $ 137 "Direction: Base Z-"
      global move_thread_flag_137=0
      thread move_thread_137():
        enter_critical
        move_thread_flag_137 = 1
        local towardsPos=calculate_point_to_move_towards(p[0.0,0.0,0.0,0.0,0.0,0.0], [0.0,0.0,-1.0], 0.067)
        movel(towardsPos, a=0.035, v=0.03)
        move_thread_flag_137 = 2
        exit_critical
      end
      move_thread_flag_137 = 0
      move_thread_han_137 = run move_thread_137()
      while (True):
        sleep(1.0E-10)
        if (move_thread_flag_137 > 1):
          join move_thread_han_137
          $ 138 "Until (distance)"
          break
        end
        sync()
      end
      $ 139 "Popup: punto contacto alanzdo"
      popup("punto contacto alanzdo", "Mensaje", False, False, blocking=True)
      $ 140 "Direction: Base Z+"
      global move_thread_flag_140=0
      thread move_thread_140():
        enter_critical
        move_thread_flag_140 = 1
        local towardsPos=calculate_point_to_move_towards(p[0.0,0.0,0.0,0.0,0.0,0.0], [0.0,0.0,1.0], 0.002)
        movel(towardsPos, a=0.005, v=0.003)
        move_thread_flag_140 = 2
        exit_critical
      end
      move_thread_flag_140 = 0
      move_thread_han_140 = run move_thread_140()
      while (True):
        sleep(1.0E-10)
        if (move_thread_flag_140 > 1):
          join move_thread_han_140
          $ 141 "Until (distance)"
          break
        end
        sync()
      end
      $ 142 "Wait: 0.3"
      sleep(0.3)
      $ 143 "Set CO[1]=Encender"
      set_configurable_digital_out(1, True)
      $ 144 "Wait: 0.3"
      sleep(0.3)
      $ 145 "Loop 3 times"
      Loop_61 = 0
      while (Loop_61 < 3):
        $ 146 "bajar≔pose_add(get_actual_tcp_pose(), bajada_broca)"
        global bajar= pose_add ( get_actual_tcp_pose (), bajada_broca)
        $ 147 "bajar" "breakAfter"
        movel(bajar, a=0.005, v=0.001)
        $ 148 "subir≔pose_sub(get_actual_tcp_pose(), bajada_broca)"
        global subir= pose_sub ( get_actual_tcp_pose (), bajada_broca)
        $ 149 "subir" "breakAfter"
        movel(subir, a=0.01, v=0.005)
        $ 150 "bajada_broca≔pose_sub(bajada_broca, bajada)"
        global bajada_broca= pose_sub (bajada_broca, bajada)
        Loop_61 = Loop_61 + 1
      end
      $ 151 "Direction: Base Z+"
      global move_thread_flag_151=0
      thread move_thread_151():
        enter_critical
        move_thread_flag_151 = 1
        local towardsPos=calculate_point_to_move_towards(p[0.0,0.0,0.0,0.0,0.0,0.0], [0.0,0.0,1.0], 0.06)
        movel(towardsPos, a=0.035, v=0.03)
        move_thread_flag_151 = 2
        exit_critical
      end
      move_thread_flag_151 = 0
      move_thread_han_151 = run move_thread_151()
      while (True):
        sleep(1.0E-10)
        if (move_thread_flag_151 > 1):
          join move_thread_han_151
          $ 152 "Until (distance)"
          break
        end
        sync()
      end
      $ 153 "Set CO[1]=Apagar"
      set_configurable_digital_out(1, False)
      $ 154 "barreno_actual≔barreno_actual+1"
      global barreno_actual=barreno_actual+1
      $ 155 "Call Quitar_broca"
      Quitar_broca()
      $ 156 "Call Poner_broca"
      Poner_broca()
    end
    $ 157 "Popup: Linea1 con chica Terminada!"
    popup("Linea1 con chica Terminada!", "Mensaje", False, False, blocking=True)
    $ 158 "Linea2"
    $ 159 "Marcar_puntos"
    $ 160 "MoveL"
    $ 161 "Home2" "breakAfter"
    movel(Home2_p, a=0.5, v=0.1)
    $ 162 "Linea2_A" "breakAfter"
    movel(Linea2_A_p, a=0.5, v=0.1)
    $ 163 "Linea2_B" "breakAfter"
    movel(Linea2_B_p, a=0.5, v=0.1)
    $ 164 "Linea2_C" "breakAfter"
    movel(Linea2_C_p, a=0.5, v=0.1)
    $ 165 "Linea2_D" "breakAfter"
    movel(Linea2_D_p, a=0.5, v=0.1)
    $ 166 "Linea2_E" "breakAfter"
    movel(Linea2_E_p, a=0.5, v=0.1)
    $ 167 "Linea2_F" "breakAfter"
    movel(Linea2_F_p, a=0.5, v=0.1)
    $ 168 "AB"
    $ 169 "'desbaste_inicial'"
    # 'desbaste_inicial'
    $ 170 "bajada_broca≔p[0,0,-0.008,0,0,0]"
    global bajada_broca=p[0,0,-0.008,0,0,0]
    $ 171 "barrenos_menos1≔8"
    global barrenos_menos1=8
    $ 172 "barreno_actual≔0"
    global barreno_actual=0
    $ 173 "Loop barreno_actual≤barrenos_menos1"
    while (barreno_actual <= barrenos_menos1):
      $ 174 "Perforacion"
      $ 175 "MoveL"
      $ 176 "internos≔interpolate_pose(Linea2_A, Linea2_B, barreno_actual/barrenos_menos1)"
      global internos= interpolate_pose (Linea2_A_p, Linea2_B_p, barreno_actual/barrenos_menos1)
      $ 177 "internos" "breakAfter"
      movel(internos, a=0.5, v=0.1)
      $ 178 "'desbaste_inicial'"
      # 'desbaste_inicial'
      $ 179 "bajada_broca≔p[0,0,-0.008,0,0,0]"
      global bajada_broca=p[0,0,-0.008,0,0,0]
      $ 180 "bajada≔p[0,0,0.008,0,0,0]"
      global bajada=p[0,0,0.008,0,0,0]
      $ 181 "Direction: Base Z-"
      global move_thread_flag_181=0
      thread move_thread_181():
        enter_critical
        move_thread_flag_181 = 1
        local towardsPos=calculate_point_to_move_towards(p[0.0,0.0,0.0,0.0,0.0,0.0], [0.0,0.0,-1.0], 0.076)
        movel(towardsPos, a=0.035, v=0.03)
        move_thread_flag_181 = 2
        exit_critical
      end
      move_thread_flag_181 = 0
      move_thread_han_181 = run move_thread_181()
      while (True):
        sleep(1.0E-10)
        if (move_thread_flag_181 > 1):
          join move_thread_han_181
          $ 182 "Until (distance)"
          break
        end
        sync()
      end
      $ 183 "Popup: punto contacto alanzdo"
      popup("punto contacto alanzdo", "Mensaje", False, False, blocking=True)
      $ 184 "Direction: Base Z+"
      global move_thread_flag_184=0
      thread move_thread_184():
        enter_critical
        move_thread_flag_184 = 1
        local towardsPos=calculate_point_to_move_towards(p[0.0,0.0,0.0,0.0,0.0,0.0], [0.0,0.0,1.0], 0.002)
        movel(towardsPos, a=0.005, v=0.003)
        move_thread_flag_184 = 2
        exit_critical
      end
      move_thread_flag_184 = 0
      move_thread_han_184 = run move_thread_184()
      while (True):
        sleep(1.0E-10)
        if (move_thread_flag_184 > 1):
          join move_thread_han_184
          $ 185 "Until (distance)"
          break
        end
        sync()
      end
      $ 186 "Wait: 0.3"
      sleep(0.3)
      $ 187 "Set CO[1]=Encender"
      set_configurable_digital_out(1, True)
      $ 188 "Wait: 0.3"
      sleep(0.3)
      $ 189 "Loop 3 times"
      Loop_63 = 0
      while (Loop_63 < 3):
        $ 190 "bajar≔pose_add(get_actual_tcp_pose(), bajada_broca)"
        global bajar= pose_add ( get_actual_tcp_pose (), bajada_broca)
        $ 191 "bajar" "breakAfter"
        movel(bajar, a=0.005, v=0.001)
        $ 192 "subir≔pose_sub(get_actual_tcp_pose(), bajada_broca)"
        global subir= pose_sub ( get_actual_tcp_pose (), bajada_broca)
        $ 193 "subir" "breakAfter"
        movel(subir, a=0.01, v=0.005)
        $ 194 "bajada_broca≔pose_sub(bajada_broca, bajada)"
        global bajada_broca= pose_sub (bajada_broca, bajada)
        Loop_63 = Loop_63 + 1
      end
      $ 195 "Direction: Base Z+"
      global move_thread_flag_195=0
      thread move_thread_195():
        enter_critical
        move_thread_flag_195 = 1
        local towardsPos=calculate_point_to_move_towards(p[0.0,0.0,0.0,0.0,0.0,0.0], [0.0,0.0,1.0], 0.06)
        movel(towardsPos, a=0.035, v=0.03)
        move_thread_flag_195 = 2
        exit_critical
      end
      move_thread_flag_195 = 0
      move_thread_han_195 = run move_thread_195()
      while (True):
        sleep(1.0E-10)
        if (move_thread_flag_195 > 1):
          join move_thread_han_195
          $ 196 "Until (distance)"
          break
        end
        sync()
      end
      $ 197 "Set CO[1]=Apagar"
      set_configurable_digital_out(1, False)
      $ 198 "barreno_actual≔barreno_actual+1"
      global barreno_actual=barreno_actual+1
      $ 199 "Call Quitar_broca"
      Quitar_broca()
      $ 200 "Call Poner_broca"
      Poner_broca()
    end
    $ 201 "CD"
    $ 202 "'desbaste_inicial'"
    # 'desbaste_inicial'
    $ 203 "bajada_broca≔p[0,0,-0.008,0,0,0]"
    global bajada_broca=p[0,0,-0.008,0,0,0]
    $ 204 "barrenos_menos1≔8"
    global barrenos_menos1=8
    $ 205 "barreno_actual≔0"
    global barreno_actual=0
    $ 206 "Loop barreno_actual≤barrenos_menos1"
    while (barreno_actual <= barrenos_menos1):
      $ 207 "Perforacion"
      $ 208 "MoveL"
      $ 209 "internos≔interpolate_pose(Linea2_C, Linea2_D, barreno_actual/barrenos_menos1)"
      global internos= interpolate_pose (Linea2_C_p, Linea2_D_p, barreno_actual/barrenos_menos1)
      $ 210 "internos" "breakAfter"
      movel(internos, a=0.5, v=0.1)
      $ 211 "'desbaste_inicial'"
      # 'desbaste_inicial'
      $ 212 "bajada_broca≔p[0,0,-0.008,0,0,0]"
      global bajada_broca=p[0,0,-0.008,0,0,0]
      $ 213 "bajada≔p[0,0,0.008,0,0,0]"
      global bajada=p[0,0,0.008,0,0,0]
      $ 214 "Direction: Base Z-"
      global move_thread_flag_214=0
      thread move_thread_214():
        enter_critical
        move_thread_flag_214 = 1
        local towardsPos=calculate_point_to_move_towards(p[0.0,0.0,0.0,0.0,0.0,0.0], [0.0,0.0,-1.0], 0.076)
        movel(towardsPos, a=0.035, v=0.03)
        move_thread_flag_214 = 2
        exit_critical
      end
      move_thread_flag_214 = 0
      move_thread_han_214 = run move_thread_214()
      while (True):
        sleep(1.0E-10)
        if (move_thread_flag_214 > 1):
          join move_thread_han_214
          $ 215 "Until (distance)"
          break
        end
        sync()
      end
      $ 216 "Popup: punto contacto alanzdo"
      popup("punto contacto alanzdo", "Mensaje", False, False, blocking=True)
      $ 217 "Direction: Base Z+"
      global move_thread_flag_217=0
      thread move_thread_217():
        enter_critical
        move_thread_flag_217 = 1
        local towardsPos=calculate_point_to_move_towards(p[0.0,0.0,0.0,0.0,0.0,0.0], [0.0,0.0,1.0], 0.002)
        movel(towardsPos, a=0.005, v=0.003)
        move_thread_flag_217 = 2
        exit_critical
      end
      move_thread_flag_217 = 0
      move_thread_han_217 = run move_thread_217()
      while (True):
        sleep(1.0E-10)
        if (move_thread_flag_217 > 1):
          join move_thread_han_217
          $ 218 "Until (distance)"
          break
        end
        sync()
      end
      $ 219 "Wait: 0.3"
      sleep(0.3)
      $ 220 "Set CO[1]=Encender"
      set_configurable_digital_out(1, True)
      $ 221 "Wait: 0.3"
      sleep(0.3)
      $ 222 "Loop 3 times"
      Loop_65 = 0
      while (Loop_65 < 3):
        $ 223 "bajar≔pose_add(get_actual_tcp_pose(), bajada_broca)"
        global bajar= pose_add ( get_actual_tcp_pose (), bajada_broca)
        $ 224 "bajar" "breakAfter"
        movel(bajar, a=0.005, v=0.001)
        $ 225 "subir≔pose_sub(get_actual_tcp_pose(), bajada_broca)"
        global subir= pose_sub ( get_actual_tcp_pose (), bajada_broca)
        $ 226 "subir" "breakAfter"
        movel(subir, a=0.01, v=0.005)
        $ 227 "bajada_broca≔pose_sub(bajada_broca, bajada)"
        global bajada_broca= pose_sub (bajada_broca, bajada)
        Loop_65 = Loop_65 + 1
      end
      $ 228 "Direction: Base Z+"
      global move_thread_flag_228=0
      thread move_thread_228():
        enter_critical
        move_thread_flag_228 = 1
        local towardsPos=calculate_point_to_move_towards(p[0.0,0.0,0.0,0.0,0.0,0.0], [0.0,0.0,1.0], 0.06)
        movel(towardsPos, a=0.035, v=0.03)
        move_thread_flag_228 = 2
        exit_critical
      end
      move_thread_flag_228 = 0
      move_thread_han_228 = run move_thread_228()
      while (True):
        sleep(1.0E-10)
        if (move_thread_flag_228 > 1):
          join move_thread_han_228
          $ 229 "Until (distance)"
          break
        end
        sync()
      end
      $ 230 "Set CO[1]=Apagar"
      set_configurable_digital_out(1, False)
      $ 231 "barreno_actual≔barreno_actual+1"
      global barreno_actual=barreno_actual+1
      $ 232 "Call Quitar_broca"
      Quitar_broca()
      $ 233 "Call Poner_broca"
      Poner_broca()
    end
    $ 234 "EF"
    $ 235 "'desbaste_inicial'"
    # 'desbaste_inicial'
    $ 236 "bajada_broca≔p[0,0,-0.008,0,0,0]"
    global bajada_broca=p[0,0,-0.008,0,0,0]
    $ 237 "barrenos_menos1≔8"
    global barrenos_menos1=8
    $ 238 "barreno_actual≔0"
    global barreno_actual=0
    $ 239 "Loop barreno_actual≤barrenos_menos1"
    while (barreno_actual <= barrenos_menos1):
      $ 240 "Perforacion"
      $ 241 "MoveL"
      $ 242 "internos≔interpolate_pose(Linea2_E, Linea2_F, barreno_actual/barrenos_menos1)"
      global internos= interpolate_pose (Linea2_E_p, Linea2_F_p, barreno_actual/barrenos_menos1)
      $ 243 "internos" "breakAfter"
      movel(internos, a=0.5, v=0.1)
      $ 244 "'desbaste_inicial'"
      # 'desbaste_inicial'
      $ 245 "bajada_broca≔p[0,0,-0.008,0,0,0]"
      global bajada_broca=p[0,0,-0.008,0,0,0]
      $ 246 "bajada≔p[0,0,0.008,0,0,0]"
      global bajada=p[0,0,0.008,0,0,0]
      $ 247 "Direction: Base Z-"
      global move_thread_flag_247=0
      thread move_thread_247():
        enter_critical
        move_thread_flag_247 = 1
        local towardsPos=calculate_point_to_move_towards(p[0.0,0.0,0.0,0.0,0.0,0.0], [0.0,0.0,-1.0], 0.076)
        movel(towardsPos, a=0.035, v=0.03)
        move_thread_flag_247 = 2
        exit_critical
      end
      move_thread_flag_247 = 0
      move_thread_han_247 = run move_thread_247()
      while (True):
        sleep(1.0E-10)
        if (move_thread_flag_247 > 1):
          join move_thread_han_247
          $ 248 "Until (distance)"
          break
        end
        sync()
      end
      $ 249 "Popup: punto contacto alanzdo"
      popup("punto contacto alanzdo", "Mensaje", False, False, blocking=True)
      $ 250 "Direction: Base Z+"
      global move_thread_flag_250=0
      thread move_thread_250():
        enter_critical
        move_thread_flag_250 = 1
        local towardsPos=calculate_point_to_move_towards(p[0.0,0.0,0.0,0.0,0.0,0.0], [0.0,0.0,1.0], 0.002)
        movel(towardsPos, a=0.005, v=0.003)
        move_thread_flag_250 = 2
        exit_critical
      end
      move_thread_flag_250 = 0
      move_thread_han_250 = run move_thread_250()
      while (True):
        sleep(1.0E-10)
        if (move_thread_flag_250 > 1):
          join move_thread_han_250
          $ 251 "Until (distance)"
          break
        end
        sync()
      end
      $ 252 "Wait: 0.3"
      sleep(0.3)
      $ 253 "Set CO[1]=Encender"
      set_configurable_digital_out(1, True)
      $ 254 "Wait: 0.3"
      sleep(0.3)
      $ 255 "Loop 3 times"
      Loop_67 = 0
      while (Loop_67 < 3):
        $ 256 "bajar≔pose_add(get_actual_tcp_pose(), bajada_broca)"
        global bajar= pose_add ( get_actual_tcp_pose (), bajada_broca)
        $ 257 "bajar" "breakAfter"
        movel(bajar, a=0.005, v=0.001)
        $ 258 "subir≔pose_sub(get_actual_tcp_pose(), bajada_broca)"
        global subir= pose_sub ( get_actual_tcp_pose (), bajada_broca)
        $ 259 "subir" "breakAfter"
        movel(subir, a=0.01, v=0.005)
        $ 260 "bajada_broca≔pose_sub(bajada_broca, bajada)"
        global bajada_broca= pose_sub (bajada_broca, bajada)
        Loop_67 = Loop_67 + 1
      end
      $ 261 "Direction: Base Z+"
      global move_thread_flag_261=0
      thread move_thread_261():
        enter_critical
        move_thread_flag_261 = 1
        local towardsPos=calculate_point_to_move_towards(p[0.0,0.0,0.0,0.0,0.0,0.0], [0.0,0.0,1.0], 0.06)
        movel(towardsPos, a=0.035, v=0.03)
        move_thread_flag_261 = 2
        exit_critical
      end
      move_thread_flag_261 = 0
      move_thread_han_261 = run move_thread_261()
      while (True):
        sleep(1.0E-10)
        if (move_thread_flag_261 > 1):
          join move_thread_han_261
          $ 262 "Until (distance)"
          break
        end
        sync()
      end
      $ 263 "Set CO[1]=Apagar"
      set_configurable_digital_out(1, False)
      $ 264 "barreno_actual≔barreno_actual+1"
      global barreno_actual=barreno_actual+1
      $ 265 "If barreno_actual>barrenos_menos1"
      if (barreno_actual>barrenos_menos1):
        $ 266 "cambiar_broca≔ True "
        global cambiar_broca=  True
      end
      $ 267 "Call Quitar_broca"
      Quitar_broca()
      $ 268 "Call Poner_broca"
      Poner_broca()
    end
    $ 269 "Popup: Linea2 con chica Terminada!"
    popup("Linea2 con chica Terminada!", "Mensaje", False, False, blocking=True)
    $ 270 "Broca_2"
    $ 271 "Linea1"
    $ 272 "Marcar_puntos"
    $ 273 "MoveL"
    $ 274 "Home2" "breakAfter"
    movel(Home2_p, a=0.5, v=0.1)
    $ 282 "Linea1_A" "breakAfter"
    movel(Linea1_A_p, a=0.5, v=0.1)
    $ 283 "Linea1_B" "breakAfter"
    movel(Linea1_B_p, a=0.5, v=0.1)
    $ 284 "Linea1_C" "breakAfter"
    movel(Linea1_C_p, a=0.5, v=0.1)
    $ 285 "Linea1_D" "breakAfter"
    movel(Linea1_D_p, a=0.5, v=0.1)
    $ 286 "Linea1_E" "breakAfter"
    movel(Linea1_E_p, a=0.5, v=0.1)
    $ 287 "Linea1_F" "breakAfter"
    movel(Linea1_F_p, a=0.5, v=0.1)
    $ 288 "AB"
    $ 289 "'desbaste_inicial'"
    # 'desbaste_inicial'
    $ 290 "bajada_broca≔p[0,0,-0.012,0,0,0]"
    global bajada_broca=p[0,0,-0.012,0,0,0]
    $ 291 "barrenos_menos1≔8"
    global barrenos_menos1=8
    $ 292 "barreno_actual≔0"
    global barreno_actual=0
    $ 293 "Loop barreno_actual≤barrenos_menos1"
    while (barreno_actual <= barrenos_menos1):
      $ 294 "Perforacion"
      $ 295 "MoveL"
      $ 296 "internos≔interpolate_pose(Linea1_A, Linea1_B, barreno_actual/barrenos_menos1)"
      global internos= interpolate_pose (Linea1_A_p, Linea1_B_p, barreno_actual/barrenos_menos1)
      $ 297 "internos" "breakAfter"
      movel(internos, a=0.5, v=0.1)
      $ 298 "'desbaste_inicial'"
      # 'desbaste_inicial'
      $ 299 "bajada_broca≔p[0,0,-0.012,0,0,0]"
      global bajada_broca=p[0,0,-0.012,0,0,0]
      $ 300 "bajada≔p[0,0,0.012,0,0,0]"
      global bajada=p[0,0,0.012,0,0,0]
      $ 301 "Direction: Base Z-"
      global move_thread_flag_301=0
      thread move_thread_301():
        enter_critical
        move_thread_flag_301 = 1
        local towardsPos=calculate_point_to_move_towards(p[0.0,0.0,0.0,0.0,0.0,0.0], [0.0,0.0,-1.0], 0.072)
        movel(towardsPos, a=0.035, v=0.03)
        move_thread_flag_301 = 2
        exit_critical
      end
      move_thread_flag_301 = 0
      move_thread_han_301 = run move_thread_301()
      while (True):
        sleep(1.0E-10)
        if (move_thread_flag_301 > 1):
          join move_thread_han_301
          $ 302 "Until (distance)"
          break
        end
        sync()
      end
      $ 303 "Popup: punto contacto alanzdo"
      popup("punto contacto alanzdo", "Mensaje", False, False, blocking=True)
      $ 304 "Direction: Base Z+"
      global move_thread_flag_304=0
      thread move_thread_304():
        enter_critical
        move_thread_flag_304 = 1
        local towardsPos=calculate_point_to_move_towards(p[0.0,0.0,0.0,0.0,0.0,0.0], [0.0,0.0,1.0], 0.002)
        movel(towardsPos, a=0.005, v=0.003)
        move_thread_flag_304 = 2
        exit_critical
      end
      move_thread_flag_304 = 0
      move_thread_han_304 = run move_thread_304()
      while (True):
        sleep(1.0E-10)
        if (move_thread_flag_304 > 1):
          join move_thread_han_304
          $ 305 "Until (distance)"
          break
        end
        sync()
      end
      $ 306 "Wait: 0.3"
      sleep(0.3)
      $ 307 "Set CO[1]=Encender"
      set_configurable_digital_out(1, True)
      $ 308 "Wait: 0.3"
      sleep(0.3)
      $ 309 "Loop 2 times"
      Loop_69 = 0
      while (Loop_69 < 2):
        $ 310 "bajar≔pose_add(get_actual_tcp_pose(), bajada_broca)"
        global bajar= pose_add ( get_actual_tcp_pose (), bajada_broca)
        $ 311 "bajar" "breakAfter"
        movel(bajar, a=0.005, v=0.001)
        $ 312 "subir≔pose_sub(get_actual_tcp_pose(), bajada_broca)"
        global subir= pose_sub ( get_actual_tcp_pose (), bajada_broca)
        $ 313 "subir" "breakAfter"
        movel(subir, a=0.01, v=0.005)
        $ 314 "bajada_broca≔pose_sub(bajada_broca, bajada)"
        global bajada_broca= pose_sub (bajada_broca, bajada)
        Loop_69 = Loop_69 + 1
      end
      $ 315 "Direction: Base Z+"
      global move_thread_flag_315=0
      thread move_thread_315():
        enter_critical
        move_thread_flag_315 = 1
        local towardsPos=calculate_point_to_move_towards(p[0.0,0.0,0.0,0.0,0.0,0.0], [0.0,0.0,1.0], 0.06)
        movel(towardsPos, a=0.035, v=0.03)
        move_thread_flag_315 = 2
        exit_critical
      end
      move_thread_flag_315 = 0
      move_thread_han_315 = run move_thread_315()
      while (True):
        sleep(1.0E-10)
        if (move_thread_flag_315 > 1):
          join move_thread_han_315
          $ 316 "Until (distance)"
          break
        end
        sync()
      end
      $ 317 "Set CO[1]=Apagar"
      set_configurable_digital_out(1, False)
      $ 318 "barreno_actual≔barreno_actual+1"
      global barreno_actual=barreno_actual+1
      $ 319 "Call Quitar_broca"
      Quitar_broca()
      $ 320 "Call Poner_broca"
      Poner_broca()
    end
    $ 321 "CD"
    $ 322 "'desbaste_inicial'"
    # 'desbaste_inicial'
    $ 323 "bajada_broca≔p[0,0,-0.012,0,0,0]"
    global bajada_broca=p[0,0,-0.012,0,0,0]
    $ 324 "barrenos_menos1≔8"
    global barrenos_menos1=8
    $ 325 "barreno_actual≔0"
    global barreno_actual=0
    $ 326 "Loop barreno_actual≤barrenos_menos1"
    while (barreno_actual <= barrenos_menos1):
      $ 327 "Perforacion"
      $ 328 "MoveL"
      $ 329 "internos≔interpolate_pose(Linea1_C, Linea1_D, barreno_actual/barrenos_menos1)"
      global internos= interpolate_pose (Linea1_C_p, Linea1_D_p, barreno_actual/barrenos_menos1)
      $ 330 "internos" "breakAfter"
      movel(internos, a=0.5, v=0.1)
      $ 331 "'desbaste_inicial'"
      # 'desbaste_inicial'
      $ 332 "bajada_broca≔p[0,0,-0.012,0,0,0]"
      global bajada_broca=p[0,0,-0.012,0,0,0]
      $ 333 "bajada≔p[0,0,0.012,0,0,0]"
      global bajada=p[0,0,0.012,0,0,0]
      $ 334 "Direction: Base Z-"
      global move_thread_flag_334=0
      thread move_thread_334():
        enter_critical
        move_thread_flag_334 = 1
        local towardsPos=calculate_point_to_move_towards(p[0.0,0.0,0.0,0.0,0.0,0.0], [0.0,0.0,-1.0], 0.072)
        movel(towardsPos, a=0.035, v=0.03)
        move_thread_flag_334 = 2
        exit_critical
      end
      move_thread_flag_334 = 0
      move_thread_han_334 = run move_thread_334()
      while (True):
        sleep(1.0E-10)
        if (move_thread_flag_334 > 1):
          join move_thread_han_334
          $ 335 "Until (distance)"
          break
        end
        sync()
      end
      $ 336 "Popup: punto contacto alanzdo"
      popup("punto contacto alanzdo", "Mensaje", False, False, blocking=True)
      $ 337 "Direction: Base Z+"
      global move_thread_flag_337=0
      thread move_thread_337():
        enter_critical
        move_thread_flag_337 = 1
        local towardsPos=calculate_point_to_move_towards(p[0.0,0.0,0.0,0.0,0.0,0.0], [0.0,0.0,1.0], 0.002)
        movel(towardsPos, a=0.005, v=0.003)
        move_thread_flag_337 = 2
        exit_critical
      end
      move_thread_flag_337 = 0
      move_thread_han_337 = run move_thread_337()
      while (True):
        sleep(1.0E-10)
        if (move_thread_flag_337 > 1):
          join move_thread_han_337
          $ 338 "Until (distance)"
          break
        end
        sync()
      end
      $ 339 "Wait: 0.3"
      sleep(0.3)
      $ 340 "Set CO[1]=Encender"
      set_configurable_digital_out(1, True)
      $ 341 "Wait: 0.3"
      sleep(0.3)
      $ 342 "Loop 2 times"
      Loop_71 = 0
      while (Loop_71 < 2):
        $ 343 "bajar≔pose_add(get_actual_tcp_pose(), bajada_broca)"
        global bajar= pose_add ( get_actual_tcp_pose (), bajada_broca)
        $ 344 "bajar" "breakAfter"
        movel(bajar, a=0.005, v=0.001)
        $ 345 "subir≔pose_sub(get_actual_tcp_pose(), bajada_broca)"
        global subir= pose_sub ( get_actual_tcp_pose (), bajada_broca)
        $ 346 "subir" "breakAfter"
        movel(subir, a=0.01, v=0.005)
        $ 347 "bajada_broca≔pose_sub(bajada_broca, bajada)"
        global bajada_broca= pose_sub (bajada_broca, bajada)
        Loop_71 = Loop_71 + 1
      end
      $ 348 "Direction: Base Z+"
      global move_thread_flag_348=0
      thread move_thread_348():
        enter_critical
        move_thread_flag_348 = 1
        local towardsPos=calculate_point_to_move_towards(p[0.0,0.0,0.0,0.0,0.0,0.0], [0.0,0.0,1.0], 0.06)
        movel(towardsPos, a=0.035, v=0.03)
        move_thread_flag_348 = 2
        exit_critical
      end
      move_thread_flag_348 = 0
      move_thread_han_348 = run move_thread_348()
      while (True):
        sleep(1.0E-10)
        if (move_thread_flag_348 > 1):
          join move_thread_han_348
          $ 349 "Until (distance)"
          break
        end
        sync()
      end
      $ 350 "Set CO[1]=Apagar"
      set_configurable_digital_out(1, False)
      $ 351 "barreno_actual≔barreno_actual+1"
      global barreno_actual=barreno_actual+1
      $ 352 "Call Quitar_broca"
      Quitar_broca()
      $ 353 "Call Poner_broca"
      Poner_broca()
    end
    $ 354 "EF"
    $ 355 "'desbaste_inicial'"
    # 'desbaste_inicial'
    $ 356 "bajada_broca≔p[0,0,-0.012,0,0,0]"
    global bajada_broca=p[0,0,-0.012,0,0,0]
    $ 357 "barrenos_menos1≔8"
    global barrenos_menos1=8
    $ 358 "barreno_actual≔0"
    global barreno_actual=0
    $ 359 "Loop barreno_actual≤barrenos_menos1"
    while (barreno_actual <= barrenos_menos1):
      $ 360 "Perforacion"
      $ 361 "MoveL"
      $ 362 "internos≔interpolate_pose(Linea1_E, Linea1_F, barreno_actual/barrenos_menos1)"
      global internos= interpolate_pose (Linea1_E_p, Linea1_F_p, barreno_actual/barrenos_menos1)
      $ 363 "internos" "breakAfter"
      movel(internos, a=0.5, v=0.1)
      $ 364 "'desbaste_inicial'"
      # 'desbaste_inicial'
      $ 365 "bajada_broca≔p[0,0,-0.012,0,0,0]"
      global bajada_broca=p[0,0,-0.012,0,0,0]
      $ 366 "bajada≔p[0,0,0.012,0,0,0]"
      global bajada=p[0,0,0.012,0,0,0]
      $ 367 "Direction: Base Z-"
      global move_thread_flag_367=0
      thread move_thread_367():
        enter_critical
        move_thread_flag_367 = 1
        local towardsPos=calculate_point_to_move_towards(p[0.0,0.0,0.0,0.0,0.0,0.0], [0.0,0.0,-1.0], 0.072)
        movel(towardsPos, a=0.035, v=0.03)
        move_thread_flag_367 = 2
        exit_critical
      end
      move_thread_flag_367 = 0
      move_thread_han_367 = run move_thread_367()
      while (True):
        sleep(1.0E-10)
        if (move_thread_flag_367 > 1):
          join move_thread_han_367
          $ 368 "Until (distance)"
          break
        end
        sync()
      end
      $ 369 "Popup: punto contacto alanzdo"
      popup("punto contacto alanzdo", "Mensaje", False, False, blocking=True)
      $ 370 "Direction: Base Z+"
      global move_thread_flag_370=0
      thread move_thread_370():
        enter_critical
        move_thread_flag_370 = 1
        local towardsPos=calculate_point_to_move_towards(p[0.0,0.0,0.0,0.0,0.0,0.0], [0.0,0.0,1.0], 0.002)
        movel(towardsPos, a=0.005, v=0.003)
        move_thread_flag_370 = 2
        exit_critical
      end
      move_thread_flag_370 = 0
      move_thread_han_370 = run move_thread_370()
      while (True):
        sleep(1.0E-10)
        if (move_thread_flag_370 > 1):
          join move_thread_han_370
          $ 371 "Until (distance)"
          break
        end
        sync()
      end
      $ 372 "Wait: 0.3"
      sleep(0.3)
      $ 373 "Set CO[1]=Encender"
      set_configurable_digital_out(1, True)
      $ 374 "Wait: 0.3"
      sleep(0.3)
      $ 375 "Loop 2 times"
      Loop_73 = 0
      while (Loop_73 < 2):
        $ 376 "bajar≔pose_add(get_actual_tcp_pose(), bajada_broca)"
        global bajar= pose_add ( get_actual_tcp_pose (), bajada_broca)
        $ 377 "bajar" "breakAfter"
        movel(bajar, a=0.005, v=0.001)
        $ 378 "subir≔pose_sub(get_actual_tcp_pose(), bajada_broca)"
        global subir= pose_sub ( get_actual_tcp_pose (), bajada_broca)
        $ 379 "subir" "breakAfter"
        movel(subir, a=0.01, v=0.005)
        $ 380 "bajada_broca≔pose_sub(bajada_broca, bajada)"
        global bajada_broca= pose_sub (bajada_broca, bajada)
        Loop_73 = Loop_73 + 1
      end
      $ 381 "Direction: Base Z+"
      global move_thread_flag_381=0
      thread move_thread_381():
        enter_critical
        move_thread_flag_381 = 1
        local towardsPos=calculate_point_to_move_towards(p[0.0,0.0,0.0,0.0,0.0,0.0], [0.0,0.0,1.0], 0.06)
        movel(towardsPos, a=0.035, v=0.03)
        move_thread_flag_381 = 2
        exit_critical
      end
      move_thread_flag_381 = 0
      move_thread_han_381 = run move_thread_381()
      while (True):
        sleep(1.0E-10)
        if (move_thread_flag_381 > 1):
          join move_thread_han_381
          $ 382 "Until (distance)"
          break
        end
        sync()
      end
      $ 383 "Set CO[1]=Apagar"
      set_configurable_digital_out(1, False)
      $ 384 "barreno_actual≔barreno_actual+1"
      global barreno_actual=barreno_actual+1
      $ 385 "Call Quitar_broca"
      Quitar_broca()
      $ 386 "Call Poner_broca"
      Poner_broca()
    end
    $ 387 "Popup: Linea1 con media Terminada!"
    popup("Linea1 con media Terminada!", "Mensaje", False, False, blocking=True)
    $ 388 "Linea2"
    $ 389 "Marcar_puntos"
    $ 390 "MoveL"
    $ 391 "Home2" "breakAfter"
    movel(Home2_p, a=0.5, v=0.1)
    $ 392 "Linea2_A" "breakAfter"
    movel(Linea2_A_p, a=0.5, v=0.1)
    $ 393 "Linea2_B" "breakAfter"
    movel(Linea2_B_p, a=0.5, v=0.1)
    $ 394 "Linea2_C" "breakAfter"
    movel(Linea2_C_p, a=0.5, v=0.1)
    $ 395 "Linea2_D" "breakAfter"
    movel(Linea2_D_p, a=0.5, v=0.1)
    $ 396 "Linea2_E" "breakAfter"
    movel(Linea2_E_p, a=0.5, v=0.1)
    $ 397 "Linea2_F" "breakAfter"
    movel(Linea2_F_p, a=0.5, v=0.1)
    $ 398 "AB"
    $ 399 "'desbaste_inicial'"
    # 'desbaste_inicial'
    $ 400 "bajada_broca≔p[0,0,-0.012,0,0,0]"
    global bajada_broca=p[0,0,-0.012,0,0,0]
    $ 401 "barrenos_menos1≔8"
    global barrenos_menos1=8
    $ 402 "barreno_actual≔0"
    global barreno_actual=0
    $ 403 "Loop barreno_actual≤barrenos_menos1"
    while (barreno_actual <= barrenos_menos1):
      $ 404 "Perforacion"
      $ 405 "MoveL"
      $ 406 "internos≔interpolate_pose(Linea2_A, Linea2_B, barreno_actual/barrenos_menos1)"
      global internos= interpolate_pose (Linea2_A_p, Linea2_B_p, barreno_actual/barrenos_menos1)
      $ 407 "internos" "breakAfter"
      movel(internos, a=0.5, v=0.1)
      $ 408 "'desbaste_inicial'"
      # 'desbaste_inicial'
      $ 409 "bajada_broca≔p[0,0,-0.012,0,0,0]"
      global bajada_broca=p[0,0,-0.012,0,0,0]
      $ 410 "bajada≔p[0,0,0.012,0,0,0]"
      global bajada=p[0,0,0.012,0,0,0]
      $ 411 "Direction: Base Z-"
      global move_thread_flag_411=0
      thread move_thread_411():
        enter_critical
        move_thread_flag_411 = 1
        local towardsPos=calculate_point_to_move_towards(p[0.0,0.0,0.0,0.0,0.0,0.0], [0.0,0.0,-1.0], 0.076)
        movel(towardsPos, a=0.035, v=0.03)
        move_thread_flag_411 = 2
        exit_critical
      end
      move_thread_flag_411 = 0
      move_thread_han_411 = run move_thread_411()
      while (True):
        sleep(1.0E-10)
        if (move_thread_flag_411 > 1):
          join move_thread_han_411
          $ 412 "Until (distance)"
          break
        end
        sync()
      end
      $ 413 "Popup: punto contacto alanzdo"
      popup("punto contacto alanzdo", "Mensaje", False, False, blocking=True)
      $ 414 "Direction: Base Z+"
      global move_thread_flag_414=0
      thread move_thread_414():
        enter_critical
        move_thread_flag_414 = 1
        local towardsPos=calculate_point_to_move_towards(p[0.0,0.0,0.0,0.0,0.0,0.0], [0.0,0.0,1.0], 0.002)
        movel(towardsPos, a=0.005, v=0.003)
        move_thread_flag_414 = 2
        exit_critical
      end
      move_thread_flag_414 = 0
      move_thread_han_414 = run move_thread_414()
      while (True):
        sleep(1.0E-10)
        if (move_thread_flag_414 > 1):
          join move_thread_han_414
          $ 415 "Until (distance)"
          break
        end
        sync()
      end
      $ 416 "Wait: 0.3"
      sleep(0.3)
      $ 417 "Set CO[1]=Encender"
      set_configurable_digital_out(1, True)
      $ 418 "Wait: 0.3"
      sleep(0.3)
      $ 419 "Loop 2 times"
      Loop_75 = 0
      while (Loop_75 < 2):
        $ 420 "bajar≔pose_add(get_actual_tcp_pose(), bajada_broca)"
        global bajar= pose_add ( get_actual_tcp_pose (), bajada_broca)
        $ 421 "bajar" "breakAfter"
        movel(bajar, a=0.005, v=0.001)
        $ 422 "subir≔pose_sub(get_actual_tcp_pose(), bajada_broca)"
        global subir= pose_sub ( get_actual_tcp_pose (), bajada_broca)
        $ 423 "subir" "breakAfter"
        movel(subir, a=0.01, v=0.005)
        $ 424 "bajada_broca≔pose_sub(bajada_broca, bajada)"
        global bajada_broca= pose_sub (bajada_broca, bajada)
        Loop_75 = Loop_75 + 1
      end
      $ 425 "Direction: Base Z+"
      global move_thread_flag_425=0
      thread move_thread_425():
        enter_critical
        move_thread_flag_425 = 1
        local towardsPos=calculate_point_to_move_towards(p[0.0,0.0,0.0,0.0,0.0,0.0], [0.0,0.0,1.0], 0.06)
        movel(towardsPos, a=0.035, v=0.03)
        move_thread_flag_425 = 2
        exit_critical
      end
      move_thread_flag_425 = 0
      move_thread_han_425 = run move_thread_425()
      while (True):
        sleep(1.0E-10)
        if (move_thread_flag_425 > 1):
          join move_thread_han_425
          $ 426 "Until (distance)"
          break
        end
        sync()
      end
      $ 427 "Set CO[1]=Apagar"
      set_configurable_digital_out(1, False)
      $ 428 "barreno_actual≔barreno_actual+1"
      global barreno_actual=barreno_actual+1
      $ 429 "Call Quitar_broca"
      Quitar_broca()
      $ 430 "Call Poner_broca"
      Poner_broca()
    end
    $ 431 "CD"
    $ 432 "'desbaste_inicial'"
    # 'desbaste_inicial'
    $ 433 "bajada_broca≔p[0,0,-0.012,0,0,0]"
    global bajada_broca=p[0,0,-0.012,0,0,0]
    $ 434 "barrenos_menos1≔8"
    global barrenos_menos1=8
    $ 435 "barreno_actual≔0"
    global barreno_actual=0
    $ 436 "Loop barreno_actual≤barrenos_menos1"
    while (barreno_actual <= barrenos_menos1):
      $ 437 "Perforacion"
      $ 438 "MoveL"
      $ 439 "internos≔interpolate_pose(Linea2_C, Linea2_D, barreno_actual/barrenos_menos1)"
      global internos= interpolate_pose (Linea2_C_p, Linea2_D_p, barreno_actual/barrenos_menos1)
      $ 440 "internos" "breakAfter"
      movel(internos, a=0.5, v=0.1)
      $ 441 "'desbaste_inicial'"
      # 'desbaste_inicial'
      $ 442 "bajada_broca≔p[0,0,-0.012,0,0,0]"
      global bajada_broca=p[0,0,-0.012,0,0,0]
      $ 443 "bajada≔p[0,0,0.012,0,0,0]"
      global bajada=p[0,0,0.012,0,0,0]
      $ 444 "Direction: Base Z-"
      global move_thread_flag_444=0
      thread move_thread_444():
        enter_critical
        move_thread_flag_444 = 1
        local towardsPos=calculate_point_to_move_towards(p[0.0,0.0,0.0,0.0,0.0,0.0], [0.0,0.0,-1.0], 0.076)
        movel(towardsPos, a=0.035, v=0.03)
        move_thread_flag_444 = 2
        exit_critical
      end
      move_thread_flag_444 = 0
      move_thread_han_444 = run move_thread_444()
      while (True):
        sleep(1.0E-10)
        if (move_thread_flag_444 > 1):
          join move_thread_han_444
          $ 445 "Until (distance)"
          break
        end
        sync()
      end
      $ 446 "Popup: punto contacto alanzdo"
      popup("punto contacto alanzdo", "Mensaje", False, False, blocking=True)
      $ 447 "Direction: Base Z+"
      global move_thread_flag_447=0
      thread move_thread_447():
        enter_critical
        move_thread_flag_447 = 1
        local towardsPos=calculate_point_to_move_towards(p[0.0,0.0,0.0,0.0,0.0,0.0], [0.0,0.0,1.0], 0.002)
        movel(towardsPos, a=0.005, v=0.003)
        move_thread_flag_447 = 2
        exit_critical
      end
      move_thread_flag_447 = 0
      move_thread_han_447 = run move_thread_447()
      while (True):
        sleep(1.0E-10)
        if (move_thread_flag_447 > 1):
          join move_thread_han_447
          $ 448 "Until (distance)"
          break
        end
        sync()
      end
      $ 449 "Wait: 0.3"
      sleep(0.3)
      $ 450 "Set CO[1]=Encender"
      set_configurable_digital_out(1, True)
      $ 451 "Wait: 0.3"
      sleep(0.3)
      $ 452 "Loop 2 times"
      Loop_78 = 0
      while (Loop_78 < 2):
        $ 453 "bajar≔pose_add(get_actual_tcp_pose(), bajada_broca)"
        global bajar= pose_add ( get_actual_tcp_pose (), bajada_broca)
        $ 454 "bajar" "breakAfter"
        movel(bajar, a=0.005, v=0.001)
        $ 455 "subir≔pose_sub(get_actual_tcp_pose(), bajada_broca)"
        global subir= pose_sub ( get_actual_tcp_pose (), bajada_broca)
        $ 456 "subir" "breakAfter"
        movel(subir, a=0.01, v=0.005)
        $ 457 "bajada_broca≔pose_sub(bajada_broca, bajada)"
        global bajada_broca= pose_sub (bajada_broca, bajada)
        Loop_78 = Loop_78 + 1
      end
      $ 458 "Direction: Base Z+"
      global move_thread_flag_458=0
      thread move_thread_458():
        enter_critical
        move_thread_flag_458 = 1
        local towardsPos=calculate_point_to_move_towards(p[0.0,0.0,0.0,0.0,0.0,0.0], [0.0,0.0,1.0], 0.06)
        movel(towardsPos, a=0.035, v=0.03)
        move_thread_flag_458 = 2
        exit_critical
      end
      move_thread_flag_458 = 0
      move_thread_han_458 = run move_thread_458()
      while (True):
        sleep(1.0E-10)
        if (move_thread_flag_458 > 1):
          join move_thread_han_458
          $ 459 "Until (distance)"
          break
        end
        sync()
      end
      $ 460 "Set CO[1]=Apagar"
      set_configurable_digital_out(1, False)
      $ 461 "barreno_actual≔barreno_actual+1"
      global barreno_actual=barreno_actual+1
      $ 462 "Call Quitar_broca"
      Quitar_broca()
      $ 463 "Call Poner_broca"
      Poner_broca()
    end
    $ 464 "EF"
    $ 465 "'desbaste_inicial'"
    # 'desbaste_inicial'
    $ 466 "bajada_broca≔p[0,0,-0.012,0,0,0]"
    global bajada_broca=p[0,0,-0.012,0,0,0]
    $ 467 "barrenos_menos1≔8"
    global barrenos_menos1=8
    $ 468 "barreno_actual≔0"
    global barreno_actual=0
    $ 469 "Loop barreno_actual≤barrenos_menos1"
    while (barreno_actual <= barrenos_menos1):
      $ 470 "Perforacion"
      $ 471 "MoveL"
      $ 472 "internos≔interpolate_pose(Linea2_E, Linea2_F, barreno_actual/barrenos_menos1)"
      global internos= interpolate_pose (Linea2_E_p, Linea2_F_p, barreno_actual/barrenos_menos1)
      $ 473 "internos" "breakAfter"
      movel(internos, a=0.5, v=0.1)
      $ 474 "'desbaste_inicial'"
      # 'desbaste_inicial'
      $ 475 "bajada_broca≔p[0,0,-0.012,0,0,0]"
      global bajada_broca=p[0,0,-0.012,0,0,0]
      $ 476 "bajada≔p[0,0,0.012,0,0,0]"
      global bajada=p[0,0,0.012,0,0,0]
      $ 477 "Direction: Base Z-"
      global move_thread_flag_477=0
      thread move_thread_477():
        enter_critical
        move_thread_flag_477 = 1
        local towardsPos=calculate_point_to_move_towards(p[0.0,0.0,0.0,0.0,0.0,0.0], [0.0,0.0,-1.0], 0.076)
        movel(towardsPos, a=0.035, v=0.03)
        move_thread_flag_477 = 2
        exit_critical
      end
      move_thread_flag_477 = 0
      move_thread_han_477 = run move_thread_477()
      while (True):
        sleep(1.0E-10)
        if (move_thread_flag_477 > 1):
          join move_thread_han_477
          $ 478 "Until (distance)"
          break
        end
        sync()
      end
      $ 479 "Popup: punto contacto alanzdo"
      popup("punto contacto alanzdo", "Mensaje", False, False, blocking=True)
      $ 480 "Direction: Base Z+"
      global move_thread_flag_480=0
      thread move_thread_480():
        enter_critical
        move_thread_flag_480 = 1
        local towardsPos=calculate_point_to_move_towards(p[0.0,0.0,0.0,0.0,0.0,0.0], [0.0,0.0,1.0], 0.002)
        movel(towardsPos, a=0.005, v=0.003)
        move_thread_flag_480 = 2
        exit_critical
      end
      move_thread_flag_480 = 0
      move_thread_han_480 = run move_thread_480()
      while (True):
        sleep(1.0E-10)
        if (move_thread_flag_480 > 1):
          join move_thread_han_480
          $ 481 "Until (distance)"
          break
        end
        sync()
      end
      $ 482 "Wait: 0.3"
      sleep(0.3)
      $ 483 "Set CO[1]=Encender"
      set_configurable_digital_out(1, True)
      $ 484 "Wait: 0.3"
      sleep(0.3)
      $ 485 "Loop 2 times"
      Loop_80 = 0
      while (Loop_80 < 2):
        $ 486 "bajar≔pose_add(get_actual_tcp_pose(), bajada_broca)"
        global bajar= pose_add ( get_actual_tcp_pose (), bajada_broca)
        $ 487 "bajar" "breakAfter"
        movel(bajar, a=0.005, v=0.001)
        $ 488 "subir≔pose_sub(get_actual_tcp_pose(), bajada_broca)"
        global subir= pose_sub ( get_actual_tcp_pose (), bajada_broca)
        $ 489 "subir" "breakAfter"
        movel(subir, a=0.01, v=0.005)
        $ 490 "bajada_broca≔pose_sub(bajada_broca, bajada)"
        global bajada_broca= pose_sub (bajada_broca, bajada)
        Loop_80 = Loop_80 + 1
      end
      $ 491 "Direction: Base Z+"
      global move_thread_flag_491=0
      thread move_thread_491():
        enter_critical
        move_thread_flag_491 = 1
        local towardsPos=calculate_point_to_move_towards(p[0.0,0.0,0.0,0.0,0.0,0.0], [0.0,0.0,1.0], 0.06)
        movel(towardsPos, a=0.035, v=0.03)
        move_thread_flag_491 = 2
        exit_critical
      end
      move_thread_flag_491 = 0
      move_thread_han_491 = run move_thread_491()
      while (True):
        sleep(1.0E-10)
        if (move_thread_flag_491 > 1):
          join move_thread_han_491
          $ 492 "Until (distance)"
          break
        end
        sync()
      end
      $ 493 "Set CO[1]=Apagar"
      set_configurable_digital_out(1, False)
      $ 494 "barreno_actual≔barreno_actual+1"
      global barreno_actual=barreno_actual+1
      $ 495 "If barreno_actual>barrenos_menos1"
      if (barreno_actual>barrenos_menos1):
        $ 496 "cambiar_broca≔ True "
        global cambiar_broca=  True
      end
      $ 497 "Call Quitar_broca"
      Quitar_broca()
      $ 498 "Call Poner_broca"
      Poner_broca()
    end
    $ 499 "Popup: Linea2 con media Terminada!"
    popup("Linea2 con media Terminada!", "Mensaje", False, False, blocking=True)
    $ 500 "Broca_3"
    $ 501 "Linea1"
    $ 502 "Marcar_puntos"
    $ 503 "MoveL"
    $ 504 "Home2" "breakAfter"
    movel(Home2_p, a=0.5, v=0.1)
    $ 505 "Linea1_A" "breakAfter"
    movel(Linea1_A_p, a=0.5, v=0.1)
    $ 506 "Linea1_B" "breakAfter"
    movel(Linea1_B_p, a=0.5, v=0.1)
    $ 507 "Linea1_C" "breakAfter"
    movel(Linea1_C_p, a=0.5, v=0.1)
    $ 508 "Linea1_D" "breakAfter"
    movel(Linea1_D_p, a=0.5, v=0.1)
    $ 509 "Linea1_E" "breakAfter"
    movel(Linea1_E_p, a=0.5, v=0.1)
    $ 510 "Linea1_F" "breakAfter"
    movel(Linea1_F_p, a=0.5, v=0.1)
    $ 511 "AB"
    $ 512 "'desbaste_inicial'"
    # 'desbaste_inicial'
    $ 513 "bajada_broca≔p[0,0,-0.012,0,0,0]"
    global bajada_broca=p[0,0,-0.012,0,0,0]
    $ 514 "barrenos_menos1≔8"
    global barrenos_menos1=8
    $ 515 "barreno_actual≔0"
    global barreno_actual=0
    $ 516 "Loop barreno_actual≤barrenos_menos1"
    while (barreno_actual <= barrenos_menos1):
      $ 517 "Perforacion"
      $ 518 "MoveL"
      $ 519 "internos≔interpolate_pose(Linea1_A, Linea1_B, barreno_actual/barrenos_menos1)"
      global internos= interpolate_pose (Linea1_A_p, Linea1_B_p, barreno_actual/barrenos_menos1)
      $ 520 "internos" "breakAfter"
      movel(internos, a=0.5, v=0.1)
      $ 521 "'desbaste_inicial'"
      # 'desbaste_inicial'
      $ 522 "bajada_broca≔p[0,0,-0.024,0,0,0]"
      global bajada_broca=p[0,0,-0.024,0,0,0]
      $ 523 "bajada≔p[0,0,0.024,0,0,0]"
      global bajada=p[0,0,0.024,0,0,0]
      $ 524 "Direction: Base Z-"
      global move_thread_flag_524=0
      thread move_thread_524():
        enter_critical
        move_thread_flag_524 = 1
        local towardsPos=calculate_point_to_move_towards(p[0.0,0.0,0.0,0.0,0.0,0.0], [0.0,0.0,-1.0], 0.072)
        movel(towardsPos, a=0.035, v=0.03)
        move_thread_flag_524 = 2
        exit_critical
      end
      move_thread_flag_524 = 0
      move_thread_han_524 = run move_thread_524()
      while (True):
        sleep(1.0E-10)
        if (move_thread_flag_524 > 1):
          join move_thread_han_524
          $ 525 "Until (distance)"
          break
        end
        sync()
      end
      $ 526 "Popup: punto contacto alanzdo"
      popup("punto contacto alanzdo", "Mensaje", False, False, blocking=True)
      $ 527 "Direction: Base Z+"
      global move_thread_flag_527=0
      thread move_thread_527():
        enter_critical
        move_thread_flag_527 = 1
        local towardsPos=calculate_point_to_move_towards(p[0.0,0.0,0.0,0.0,0.0,0.0], [0.0,0.0,1.0], 0.002)
        movel(towardsPos, a=0.005, v=0.003)
        move_thread_flag_527 = 2
        exit_critical
      end
      move_thread_flag_527 = 0
      move_thread_han_527 = run move_thread_527()
      while (True):
        sleep(1.0E-10)
        if (move_thread_flag_527 > 1):
          join move_thread_han_527
          $ 528 "Until (distance)"
          break
        end
        sync()
      end
      $ 529 "Wait: 0.3"
      sleep(0.3)
      $ 530 "Set CO[1]=Encender"
      set_configurable_digital_out(1, True)
      $ 531 "Wait: 0.3"
      sleep(0.3)
      $ 532 "Loop 1 times"
      Loop_82 = 0
      while (Loop_82 < 1):
        $ 533 "bajar≔pose_add(get_actual_tcp_pose(), bajada_broca)"
        global bajar= pose_add ( get_actual_tcp_pose (), bajada_broca)
        $ 534 "bajar" "breakAfter"
        movel(bajar, a=0.005, v=0.001)
        $ 535 "subir≔pose_sub(get_actual_tcp_pose(), bajada_broca)"
        global subir= pose_sub ( get_actual_tcp_pose (), bajada_broca)
        $ 536 "subir" "breakAfter"
        movel(subir, a=0.01, v=0.005)
        $ 537 "bajada_broca≔pose_sub(bajada_broca, bajada)"
        global bajada_broca= pose_sub (bajada_broca, bajada)
        Loop_82 = Loop_82 + 1
      end
